C07315=1163.961,-99.989,-42.259,178.914,5.840,149.363
C07316=1163.967,-100.239,-42.250,178.911,5.839,149.364
C07317=1163.973,-100.489,-42.240,178.909,5.838,149.364
C07318=1163.977,-100.739,-42.231,178.907,5.838,149.365
C07319=1163.983,-100.989,-42.221,178.905,5.838,149.365
C07320=1163.988,-101.238,-42.212,178.903,5.838,149.366
C07321=1163.993,-101.488,-42.203,178.901,5.837,149.367
C07322=1163.999,-101.738,-42.193,178.899,5.837,149.367
C07323=1164.005,-102.010,-42.183,178.896,5.837,149.368
C07324=1164.011,-102.281,-42.173,178.894,5.836,149.368
C07325=1164.016,-102.553,-42.163,178.892,5.836,149.369
C07326=1164.022,-102.825,-42.153,178.890,5.836,149.370
C07327=1164.028,-103.075,-42.143,178.887,5.835,149.370
C07328=1164.033,-103.325,-42.134,178.885,5.835,149.371
C07329=1164.038,-103.574,-42.125,178.883,5.835,149.371
C07330=1164.044,-103.824,-42.115,178.881,5.834,149.372
C07331=1164.049,-104.074,-42.106,178.879,5.834,149.372
C07332=1164.054,-104.323,-42.097,178.877,5.834,149.373
C07333=1164.060,-104.574,-42.087,178.875,5.834,149.374
C07334=1164.065,-104.823,-42.078,178.873,5.833,149.374
C07335=1164.070,-105.073,-42.069,178.870,5.833,149.375
C07336=1164.076,-105.323,-42.059,178.868,5.833,149.375
C07337=1164.081,-105.573,-42.050,178.866,5.832,149.376
C07338=1164.086,-105.823,-42.041,178.864,5.833,149.376
C07339=1164.092,-106.073,-42.032,178.862,5.832,149.377
C07340=1164.097,-106.322,-42.022,178.860,5.832,149.377
C07341=1164.102,-106.572,-42.013,178.858,5.831,149.378
C07342=1164.107,-106.822,-42.004,178.856,5.831,149.379
C07343=1164.113,-107.072,-41.995,178.854,5.831,149.379
C07344=1164.118,-107.321,-41.985,178.851,5.830,149.380
C07345=1164.123,-107.571,-41.976,178.850,5.830,149.380
C07346=1164.128,-107.821,-41.968,178.847,5.830,149.381
C07347=1164.134,-108.071,-41.958,178.845,5.830,149.382
C07348=1164.140,-108.320,-41.950,178.843,5.829,149.382
C07349=1164.145,-108.570,-41.941,178.842,5.829,149.383
C07350=1164.150,-108.819,-41.931,178.839,5.829,149.383
C07351=1164.156,-109.069,-41.922,178.837,5.828,149.384
C07352=1164.161,-109.319,-41.913,178.835,5.828,149.384
C07353=1164.166,-109.569,-41.904,178.832,5.828,149.385
C07354=1164.171,-109.819,-41.895,178.831,5.828,149.385
C07355=1164.177,-110.069,-41.885,178.829,5.827,149.386
C07356=1164.182,-110.319,-41.876,178.827,5.827,149.387
C07357=1164.187,-110.568,-41.867,178.824,5.827,149.387
C07358=1164.192,-110.818,-41.858,178.823,5.827,149.388
C07359=1164.197,-111.068,-41.849,178.820,5.826,149.388
C07360=1164.204,-111.317,-41.840,178.819,5.826,149.389
C07361=1164.209,-111.567,-41.831,178.816,5.826,149.389
C07362=1164.214,-111.817,-41.822,178.814,5.825,149.390
C07363=1164.219,-112.067,-41.813,178.812,5.825,149.390
C07364=1164.225,-112.317,-41.804,178.810,5.824,149.391
C07365=1164.230,-112.567,-41.795,178.808,5.825,149.392
C07366=1164.236,-112.817,-41.786,178.806,5.824,149.392
C07367=1164.241,-113.067,-41.777,178.804,5.824,149.393
C07368=1164.246,-113.315,-41.768,178.802,5.823,149.393
C07369=1164.251,-113.565,-41.759,178.800,5.824,149.394
C07370=1164.257,-113.815,-41.750,178.798,5.823,149.394
C07371=1164.263,-114.065,-41.741,178.796,5.823,149.395
C07372=1164.268,-114.315,-41.732,178.793,5.823,149.396
C07373=1164.273,-114.565,-41.723,178.791,5.822,149.396
C07374=1164.278,-114.814,-41.714,178.789,5.822,149.396
C07375=1164.284,-115.064,-41.705,178.787,5.822,149.397
C07376=1164.289,-115.313,-41.696,178.785,5.822,149.398
C07377=1164.294,-115.563,-41.687,178.783,5.821,149.398
C07378=1164.299,-115.813,-41.679,178.781,5.821,149.399
C07379=1164.305,-116.063,-41.669,178.779,5.821,149.399
C07380=1164.310,-116.313,-41.660,178.777,5.821,149.400
C07381=1164.316,-116.562,-41.652,178.775,5.820,149.400
C07382=1164.322,-116.813,-41.643,178.773,5.820,149.401
C07383=1164.327,-117.063,-41.635,178.771,5.819,149.402
C07384=1164.332,-117.313,-41.626,178.769,5.820,149.402
C07385=1164.337,-117.562,-41.617,178.766,5.819,149.403
C07386=1164.342,-117.812,-41.608,178.765,5.819,149.403
C07387=1164.348,-118.061,-41.599,178.763,5.818,149.404
C07388=1164.353,-118.311,-41.590,178.761,5.818,149.404
C07389=1164.358,-118.561,-41.582,178.758,5.818,149.405
C07390=1164.364,-118.811,-41.573,178.757,5.818,149.405
C07391=1164.369,-119.061,-41.563,178.754,5.817,149.406
C07392=1164.375,-119.310,-41.555,178.752,5.818,149.407
C07393=1164.380,-119.560,-41.546,178.750,5.817,149.407
C07394=1164.386,-119.810,-41.537,178.748,5.816,149.408
C07395=1164.391,-120.060,-41.529,178.746,5.816,149.408
C07396=1164.396,-120.310,-41.520,178.744,5.816,149.409
C07397=1164.402,-120.559,-41.511,178.742,5.816,149.409
C07398=1164.407,-120.809,-41.502,178.740,5.815,149.410
C07399=1164.412,-121.059,-41.493,178.738,5.815,149.410
C07400=1164.417,-121.309,-41.485,178.736,5.815,149.411
C07401=1164.423,-121.558,-41.476,178.734,5.815,149.411
C07402=1164.429,-121.809,-41.468,178.732,5.814,149.412
C07403=1164.434,-122.058,-41.459,178.730,5.815,149.413
C07404=1164.439,-122.308,-41.450,178.728,5.814,149.413
C07405=1164.444,-122.558,-41.441,178.726,5.814,149.414
C07406=1164.450,-122.807,-41.433,178.724,5.813,149.414
C07407=1164.455,-123.058,-41.424,178.722,5.814,149.415
C07408=1164.461,-123.308,-41.416,178.720,5.813,149.415
C07409=1164.466,-123.557,-41.407,178.718,5.813,149.416
C07410=1164.471,-123.807,-41.398,178.716,5.812,149.416
C07411=1164.477,-124.056,-41.389,178.714,5.812,149.417
C07412=1164.482,-124.307,-41.381,178.711,5.812,149.418
C07413=1164.487,-124.556,-41.373,178.710,5.812,149.418
C07414=1164.492,-124.806,-41.364,178.708,5.811,149.418
C07415=1164.497,-125.055,-41.355,178.706,5.811,149.419
C07416=1164.503,-125.306,-41.347,178.703,5.811,149.420
C07417=1164.509,-125.555,-41.339,178.702,5.811,149.420
C07418=1164.514,-125.805,-41.330,178.700,5.810,149.421
C07419=1164.519,-126.055,-41.321,178.698,5.810,149.421
C07420=1164.525,-126.305,-41.313,178.695,5.810,149.422
C07421=1164.530,-126.554,-41.304,178.694,5.810,149.422
C07422=1164.535,-126.804,-41.295,178.692,5.809,149.423
C07423=1164.541,-127.055,-41.287,178.689,5.809,149.424
C07424=1164.547,-127.304,-41.278,178.687,5.809,149.424
C07425=1164.552,-127.554,-41.270,178.686,5.809,149.425
C07426=1164.557,-127.804,-41.262,178.683,5.808,149.425
C07427=1164.136,-127.815,-41.303,178.680,5.812,149.427
C07428=1164.130,-127.565,-41.311,178.682,5.812,149.426
C07429=1164.125,-127.315,-41.320,178.684,5.813,149.426
C07430=1164.119,-127.066,-41.329,178.686,5.812,149.425
C07431=1164.114,-126.815,-41.337,178.688,5.813,149.425
C07432=1164.109,-126.565,-41.346,178.690,5.813,149.424
C07433=1164.104,-126.316,-41.354,178.692,5.814,149.424
C07434=1164.098,-126.066,-41.362,178.694,5.813,149.423
C07435=1164.093,-125.816,-41.371,178.696,5.814,149.422
C07436=1164.088,-125.566,-41.380,178.698,5.814,149.422
C07437=1164.082,-125.317,-41.388,178.700,5.815,149.422
C07438=1164.077,-125.067,-41.396,178.702,5.815,149.421
C07439=1164.072,-124.817,-41.405,178.704,5.815,149.420
C07440=1164.066,-124.568,-41.414,178.706,5.815,149.420
C07441=1164.061,-124.318,-41.423,178.708,5.816,149.419
C07442=1164.055,-124.067,-41.431,178.710,5.816,149.419
C07443=1164.050,-123.818,-41.440,178.712,5.816,149.418
C07444=1164.044,-123.568,-41.448,178.714,5.816,149.418
C07445=1164.039,-123.319,-41.457,178.716,5.817,149.417
C07446=1164.034,-123.069,-41.466,178.718,5.817,149.417
C07447=1164.028,-122.818,-41.474,178.721,5.817,149.416
C07448=1164.023,-122.569,-41.483,178.722,5.817,149.415
C07449=1164.017,-122.319,-41.492,178.724,5.818,149.415
C07450=1164.012,-122.069,-41.501,178.726,5.817,149.414
C07451=1164.007,-121.819,-41.510,178.729,5.818,149.414
C07452=1164.001,-121.570,-41.517,178.730,5.818,149.413
C07453=1163.996,-121.320,-41.526,178.732,5.819,149.413
C07454=1163.991,-121.070,-41.535,178.734,5.818,149.412
C07455=1163.986,-120.820,-41.544,178.737,5.819,149.412
C07456=1163.980,-120.570,-41.553,178.738,5.819,149.411
C07457=1163.975,-120.321,-41.562,178.740,5.820,149.411
C07458=1163.969,-120.071,-41.570,178.743,5.820,149.410
C07459=1163.964,-119.821,-41.579,178.745,5.820,149.409
C07460=1163.959,-119.571,-41.587,178.746,5.820,149.409
C07461=1163.953,-119.322,-41.596,178.749,5.821,149.408
C07462=1163.948,-119.072,-41.605,178.751,5.821,149.408
C07463=1163.943,-118.822,-41.614,178.753,5.821,149.407
C07464=1163.938,-118.572,-41.623,178.754,5.821,149.407
C07465=1163.932,-118.322,-41.632,178.757,5.822,149.406
C07466=1163.927,-118.073,-41.641,178.759,5.822,149.406
C07467=1163.921,-117.823,-41.649,178.761,5.822,149.405
C07468=1163.916,-117.574,-41.658,178.762,5.822,149.405
C07469=1163.911,-117.323,-41.666,178.765,5.823,149.404
C07470=1163.906,-117.073,-41.675,178.767,5.824,149.403
C07471=1163.900,-116.823,-41.684,178.769,5.823,149.403
C07472=1163.894,-116.574,-41.693,178.772,5.824,149.402
C07473=1163.889,-116.324,-41.702,178.773,5.824,149.402
C07474=1163.884,-116.074,-41.711,178.775,5.825,149.401
C07475=1163.878,-115.824,-41.720,178.777,5.825,149.401
C07476=1163.873,-115.575,-41.729,178.780,5.825,149.400
C07477=1163.868,-115.325,-41.738,178.781,5.825,149.400
C07478=1163.862,-115.076,-41.746,178.783,5.826,149.399
C07479=1163.857,-114.826,-41.755,178.786,5.825,149.398
C07480=1163.851,-114.576,-41.764,178.788,5.826,149.398
C07481=1163.846,-114.326,-41.773,178.789,5.826,149.397
C07482=1163.841,-114.076,-41.782,178.792,5.826,149.397
C07483=1163.836,-113.826,-41.791,178.794,5.826,149.396
C07484=1163.831,-113.576,-41.800,178.796,5.827,149.396
C07485=1163.825,-113.327,-41.809,178.797,5.827,149.395
C07486=1163.820,-113.077,-41.817,178.800,5.827,149.394
C07487=1163.814,-112.827,-41.827,178.802,5.828,149.394
C07488=1163.809,-112.577,-41.836,178.804,5.828,149.393
C07489=1163.803,-112.327,-41.845,178.807,5.829,149.393
C07490=1163.799,-112.078,-41.854,178.808,5.828,149.392
C07491=1163.793,-111.828,-41.863,178.810,5.829,149.392
C07492=1163.788,-111.578,-41.872,178.812,5.829,149.391
C07493=1163.782,-111.329,-41.881,178.815,5.830,149.391
C07494=1163.777,-111.079,-41.890,178.816,5.830,149.390
C07495=1163.771,-110.829,-41.899,178.819,5.830,149.389
C07496=1163.766,-110.579,-41.908,178.821,5.830,149.389
C07497=1163.761,-110.329,-41.917,178.823,5.831,149.388
C07498=1163.755,-110.079,-41.926,178.825,5.831,149.388
C07499=1163.750,-109.829,-41.935,178.827,5.831,149.387
C07500=1163.745,-109.580,-41.945,178.829,5.832,149.387
C07501=1163.740,-109.330,-41.954,178.831,5.832,149.386
C07502=1163.734,-109.080,-41.963,178.833,5.832,149.386
C07503=1163.729,-108.830,-41.972,178.835,5.832,149.385
C07504=1163.723,-108.581,-41.981,178.837,5.833,149.385
C07505=1163.718,-108.331,-41.990,178.839,5.832,149.384
C07506=1163.712,-108.082,-42.000,178.842,5.833,149.383
C07507=1163.707,-107.832,-42.009,178.844,5.834,149.383
C07508=1163.702,-107.582,-42.018,178.846,5.834,149.382
C07509=1163.697,-107.332,-42.027,178.848,5.834,149.382
C07510=1163.691,-107.082,-42.036,178.850,5.834,149.381
C07511=1163.686,-106.833,-42.046,178.852,5.835,149.380
C07512=1163.681,-106.583,-42.055,178.854,5.835,149.380
C07513=1163.676,-106.333,-42.063,178.856,5.835,149.380
C07514=1163.670,-106.083,-42.073,178.859,5.836,149.379
C07515=1163.665,-105.833,-42.082,178.860,5.836,149.378
C07516=1163.660,-105.584,-42.091,178.863,5.837,149.378
C07517=1163.654,-105.334,-42.101,178.865,5.836,149.377
C07518=1163.649,-105.084,-42.110,178.867,5.837,149.377
C07519=1163.644,-104.834,-42.119,178.868,5.837,149.376
C07520=1163.639,-104.585,-42.128,178.871,5.837,149.375
C07521=1163.633,-104.335,-42.138,178.873,5.838,149.375
C07522=1163.628,-104.085,-42.147,178.875,5.838,149.374
C07523=1163.623,-103.836,-42.156,178.878,5.838,149.374
C07524=1163.617,-103.585,-42.166,178.879,5.838,149.373
C07525=1163.612,-103.336,-42.175,178.882,5.839,149.373
C07526=1163.607,-103.086,-42.184,178.883,5.839,149.372
C07527=1163.601,-102.836,-42.194,178.886,5.839,149.372
C07528=1163.596,-102.564,-42.204,178.888,5.840,149.371
C07529=1163.589,-102.292,-42.213,178.890,5.840,149.370
C07530=1163.584,-102.020,-42.223,178.893,5.840,149.370
C07531=1163.577,-101.748,-42.234,178.895,5.841,149.369
C07532=1163.573,-101.499,-42.244,178.897,5.840,149.368
C07533=1163.567,-101.249,-42.253,178.899,5.841,149.368
C07534=1163.561,-100.999,-42.262,178.902,5.842,149.367
C07535=1163.557,-100.750,-42.272,178.903,5.842,149.367
C07536=1163.551,-100.500,-42.281,178.905,5.842,149.366
C07537=1163.546,-100.250,-42.290,178.908,5.842,149.366
C07538=1163.541,-100.001,-42.300,178.910,5.843,149.365
C07539=1163.535,-99.750,-42.309,178.912,5.844,149.365
C07540=1163.530,-99.501,-42.319,178.914,5.843,149.364
C07541=1163.525,-99.251,-42.328,178.916,5.844,149.363
C07542=1163.519,-99.001,-42.337,178.918,5.843,149.363
C07543=1163.514,-98.752,-42.347,178.920,5.844,149.362
C07544=1163.508,-98.502,-42.356,178.923,5.845,149.362
C07545=1163.504,-98.252,-42.366,178.925,5.845,149.361
C07546=1163.498,-98.002,-42.376,178.927,5.845,149.361
C07547=1163.493,-97.752,-42.386,178.929,5.845,149.360
C07548=1163.487,-97.502,-42.395,178.931,5.846,149.359
C07549=1163.482,-97.253,-42.405,178.933,5.846,149.359
C07550=1163.476,-97.003,-42.414,178.935,5.846,149.358
C07551=1163.471,-96.753,-42.423,178.938,5.847,149.358
C07552=1163.466,-96.504,-42.433,178.939,5.847,149.357
C07553=1163.460,-96.254,-42.442,178.942,5.847,149.356
C07554=1163.456,-96.004,-42.452,178.944,5.848,149.356
C07555=1163.450,-95.754,-42.461,178.946,5.848,149.356
C07556=1163.445,-95.505,-42.471,178.948,5.848,149.355
C07557=1163.439,-95.255,-42.480,178.950,5.848,149.354
C07558=1163.435,-95.005,-42.490,178.953,5.849,149.354
C07559=1163.429,-94.755,-42.500,178.955,5.849,149.353
C07560=1163.424,-94.505,-42.509,178.956,5.849,149.353
C07561=1163.418,-94.256,-42.520,178.959,5.850,149.352
C07562=1163.413,-94.006,-42.529,178.961,5.850,149.351
C07563=1163.408,-93.757,-42.539,178.963,5.850,149.351
C07564=1163.402,-93.506,-42.548,178.966,5.851,149.350
C07565=1163.397,-93.257,-42.558,178.967,5.851,149.350
C07566=1163.391,-93.007,-42.567,178.970,5.851,149.349
C07567=1163.387,-92.757,-42.577,178.972,5.852,149.349
C07568=1163.381,-92.507,-42.587,178.974,5.852,149.348
C07569=1163.376,-92.258,-42.596,178.976,5.852,149.347
C07570=1163.370,-92.008,-42.607,178.978,5.852,149.347
C07571=1163.365,-91.758,-42.616,178.981,5.853,149.346
C07572=1163.359,-91.509,-42.626,178.983,5.854,149.346
C07573=1163.354,-91.258,-42.636,178.985,5.853,149.345
C07574=1163.349,-91.009,-42.645,178.987,5.854,149.344
C07575=1163.344,-90.759,-42.655,178.989,5.855,149.344
C07576=1163.339,-90.509,-42.664,178.991,5.854,149.343
C07577=1163.333,-90.260,-42.675,178.994,5.855,149.343
C07578=1163.328,-90.010,-42.684,178.996,5.855,149.342
C07579=1163.323,-89.760,-42.694,178.998,5.855,149.342
C07580=1163.317,-89.510,-42.704,179.000,5.856,149.341
C07581=1163.312,-89.261,-42.714,179.002,5.856,149.340
C07582=1163.306,-89.011,-42.723,179.004,5.857,149.340
C07583=1163.301,-88.761,-42.734,179.007,5.857,149.339
C07584=1163.296,-88.512,-42.743,179.009,5.857,149.339
C07585=1163.291,-88.262,-42.754,179.011,5.858,149.338
C07586=1163.286,-88.012,-42.763,179.013,5.857,149.338
C07587=1163.280,-87.762,-42.773,179.015,5.858,149.337
C07588=1163.275,-87.513,-42.783,179.018,5.858,149.336
C07589=1163.269,-87.263,-42.792,179.019,5.858,149.336
C07590=1163.264,-87.013,-42.803,179.022,5.859,149.335
C07591=1163.259,-86.763,-42.813,179.024,5.860,149.335
C07592=1163.254,-86.514,-42.822,179.026,5.860,149.334
C07593=1163.248,-86.264,-42.832,179.028,5.860,149.333
C07594=1163.243,-86.013,-42.842,179.031,5.861,149.333
C07595=1163.238,-85.764,-42.852,179.033,5.860,149.332
C07596=1163.233,-85.515,-42.862,179.035,5.861,149.332
C07597=1163.227,-85.264,-42.872,179.037,5.862,149.331
C07598=1163.222,-85.015,-42.882,179.039,5.861,149.331
C07599=1163.217,-84.765,-42.892,179.041,5.862,149.330
C07600=1163.211,-84.515,-42.902,179.044,5.863,149.329
C07601=1163.206,-84.266,-42.912,179.046,5.863,149.329
C07602=1163.201,-84.016,-42.922,179.048,5.863,149.328
C07603=1163.195,-83.766,-42.932,179.050,5.864,149.328
C07604=1163.190,-83.516,-42.942,179.052,5.864,149.327
C07605=1163.185,-83.267,-42.952,179.055,5.864,149.327
C07606=1163.180,-83.017,-42.962,179.057,5.865,149.326
C07607=1163.174,-82.767,-42.972,179.059,5.865,149.325
C07608=1163.169,-82.518,-42.983,179.061,5.865,149.325
C07609=1163.164,-82.268,-42.992,179.064,5.866,149.324
C07610=1163.159,-82.018,-43.002,179.065,5.866,149.324
C07611=1163.153,-81.768,-43.012,179.068,5.866,149.323
C07612=1163.147,-81.519,-43.023,179.070,5.867,149.323
C07613=1163.143,-81.269,-43.033,179.072,5.867,149.322
C07614=1163.138,-81.019,-43.043,179.075,5.867,149.321
C07615=1163.132,-80.769,-43.053,179.077,5.868,149.321
C07616=1163.126,-80.520,-43.063,179.079,5.868,149.320
C07617=1163.122,-80.270,-43.073,179.081,5.868,149.320
C07618=1163.117,-80.020,-43.083,179.084,5.869,149.319
C07619=1163.111,-79.771,-43.094,179.085,5.869,149.318
C07620=1163.106,-79.520,-43.103,179.088,5.870,149.318
C07621=1163.100,-79.271,-43.114,179.090,5.870,149.317
C07622=1163.094,-79.021,-43.124,179.092,5.870,149.317
C07623=1163.090,-78.771,-43.134,179.094,5.870,149.316
C07624=1163.085,-78.522,-43.144,179.097,5.871,149.316
C07625=1163.079,-78.272,-43.154,179.099,5.871,149.315
C07626=1163.074,-78.022,-43.165,179.101,5.871,149.314
C07627=1163.068,-77.772,-43.175,179.104,5.872,149.314
C07628=1163.063,-77.523,-43.185,179.105,5.872,149.313
C07629=1163.059,-77.273,-43.195,179.107,5.873,149.313
C07630=1163.053,-77.023,-43.205,179.110,5.873,149.312
C07631=1163.047,-76.774,-43.216,179.112,5.873,149.312
C07632=1163.041,-76.502,-43.227,179.114,5.873,149.311
C07633=1163.036,-76.231,-43.238,179.117,5.874,149.310
C07634=1163.030,-75.960,-43.249,179.119,5.875,149.310
C07635=1163.025,-75.689,-43.261,179.122,5.875,149.309
C07636=1163.019,-75.440,-43.271,179.124,5.875,149.308
C07637=1163.014,-75.189,-43.282,179.126,5.875,149.308
C07638=1163.009,-74.940,-43.292,179.128,5.876,149.307
C07639=1163.003,-74.690,-43.302,179.131,5.877,149.307
C07640=1162.998,-74.440,-43.313,179.133,5.877,149.306
C07641=1162.992,-74.190,-43.323,179.135,5.877,149.305
C07642=1162.987,-73.940,-43.333,179.137,5.878,149.305
C07643=1162.982,-73.691,-43.344,179.139,5.877,149.304
C07644=1162.976,-73.441,-43.354,179.142,5.878,149.304
C07645=1162.971,-73.191,-43.364,179.144,5.878,149.303
C07646=1162.967,-72.942,-43.375,179.146,5.878,149.303
C07647=1162.961,-72.693,-43.385,179.149,5.879,149.302
C07648=1162.956,-72.442,-43.396,179.151,5.880,149.301
C07649=1162.951,-72.193,-43.406,179.153,5.880,149.301
C07650=1162.946,-71.943,-43.416,179.155,5.880,149.300
C07651=1162.940,-71.693,-43.427,179.157,5.881,149.300
C07652=1162.935,-71.443,-43.437,179.160,5.881,149.299
C07653=1162.930,-71.194,-43.448,179.162,5.881,149.298
C07654=1162.924,-70.944,-43.458,179.164,5.882,149.298
C07655=1162.919,-70.694,-43.469,179.166,5.882,149.297
C07656=1162.913,-70.445,-43.479,179.169,5.883,149.297
C07657=1162.908,-70.194,-43.490,179.171,5.883,149.296
C07658=1162.903,-69.945,-43.501,179.173,5.883,149.295
C07659=1162.898,-69.695,-43.511,179.176,5.884,149.295
C07660=1162.893,-69.446,-43.521,179.178,5.884,149.294
C07661=1162.887,-69.196,-43.532,179.180,5.884,149.294
C07662=1162.882,-68.947,-43.543,179.182,5.885,149.293
C07663=1162.877,-68.697,-43.553,179.185,5.885,149.293
C07664=1162.872,-68.447,-43.564,179.187,5.885,149.292
C07665=1162.866,-68.197,-43.574,179.189,5.886,149.291
C07666=1162.861,-67.948,-43.585,179.192,5.886,149.291
C07667=1162.855,-67.698,-43.596,179.194,5.887,149.290
C07668=1162.850,-67.447,-43.606,179.195,5.887,149.290
C07669=1162.844,-67.198,-43.617,179.198,5.887,149.289
C07670=1162.840,-66.948,-43.628,179.200,5.888,149.288
C07671=1162.834,-66.699,-43.638,179.202,5.888,149.288
C07672=1162.829,-66.449,-43.649,179.204,5.889,149.287
C07673=1162.824,-66.200,-43.660,179.207,5.889,149.287
C07674=1162.819,-65.949,-43.670,179.209,5.890,149.286
C07675=1162.813,-65.700,-43.680,179.211,5.889,149.285
C07676=1162.809,-65.450,-43.692,179.214,5.890,149.285
C07677=1162.803,-65.201,-43.702,179.216,5.891,149.284
C07678=1162.798,-64.950,-43.713,179.218,5.891,149.284
C07679=1162.793,-64.701,-43.723,179.221,5.891,149.283
C07680=1162.787,-64.451,-43.735,179.223,5.892,149.283
C07681=1162.782,-64.202,-43.746,179.225,5.892,149.282
C07682=1162.777,-63.952,-43.756,179.228,5.893,149.281
C07683=1162.771,-63.702,-43.766,179.230,5.893,149.281
C07684=1162.766,-63.453,-43.778,179.232,5.893,149.280
C07685=1162.761,-63.203,-43.788,179.235,5.894,149.279
C07686=1162.756,-62.953,-43.799,179.237,5.895,149.279
C07687=1162.750,-62.704,-43.810,179.239,5.894,149.278
C07688=1162.745,-62.453,-43.821,179.241,5.895,149.278
C07689=1162.740,-62.204,-43.832,179.244,5.895,149.277
C07690=1162.734,-61.954,-43.842,179.246,5.896,149.277
C07691=1162.730,-61.705,-43.853,179.248,5.896,149.276
C07692=1162.724,-61.455,-43.864,179.250,5.897,149.275
C07693=1162.719,-61.205,-43.875,179.253,5.897,149.275
C07694=1162.713,-60.955,-43.886,179.255,5.898,149.274
C07695=1162.708,-60.706,-43.897,179.257,5.897,149.274
C07696=1162.703,-60.456,-43.907,179.259,5.898,149.273
C07697=1162.698,-60.207,-43.918,179.262,5.899,149.272
C07698=1162.693,-59.956,-43.929,179.264,5.899,149.272
C07699=1162.687,-59.707,-43.940,179.267,5.900,149.271
C07700=1162.682,-59.457,-43.951,179.268,5.900,149.271
C07701=1162.677,-59.207,-43.962,179.271,5.900,149.270
C07702=1162.672,-58.958,-43.973,179.273,5.901,149.270
C07703=1162.666,-58.708,-43.984,179.276,5.901,149.269
C07704=1162.661,-58.458,-43.995,179.277,5.901,149.268
C07705=1162.656,-58.209,-44.006,179.280,5.902,149.268
C07706=1162.651,-57.958,-44.017,179.282,5.903,149.267
C07707=1162.645,-57.709,-44.028,179.285,5.903,149.266
C07708=1162.640,-57.460,-44.039,179.287,5.903,149.266
C07709=1162.635,-57.210,-44.050,179.289,5.903,149.265
C07710=1162.630,-56.960,-44.061,179.291,5.904,149.265
C07711=1162.624,-56.710,-44.072,179.294,5.905,149.264
C07712=1162.619,-56.461,-44.083,179.296,5.905,149.264
C07713=1162.614,-56.211,-44.094,179.298,5.905,149.263
C07714=1162.609,-55.961,-44.105,179.300,5.906,149.262
C07715=1162.603,-55.712,-44.116,179.303,5.906,149.262
C07716=1162.598,-55.462,-44.127,179.305,5.907,149.261
C07717=1162.594,-55.212,-44.138,179.308,5.907,149.261
C07718=1162.588,-54.963,-44.150,179.310,5.907,149.260
C07719=1162.583,-54.712,-44.160,179.312,5.908,149.259
C07720=1162.578,-54.463,-44.172,179.314,5.909,149.259
C07721=1162.572,-54.214,-44.183,179.317,5.909,149.258
C07722=1162.567,-53.963,-44.194,179.319,5.910,149.258
C07723=1162.562,-53.714,-44.205,179.321,5.909,149.257
C07724=1162.556,-53.465,-44.216,179.324,5.910,149.257
C07725=1162.551,-53.215,-44.228,179.326,5.911,149.256
C07726=1162.546,-52.965,-44.238,179.328,5.911,149.255
C07727=1162.540,-52.715,-44.250,179.331,5.912,149.255
C07728=1162.536,-52.466,-44.261,179.333,5.912,149.254
C07729=1162.531,-52.216,-44.272,179.335,5.912,149.253
C07730=1162.525,-51.966,-44.284,179.338,5.913,149.253
C07731=1162.520,-51.717,-44.295,179.340,5.913,149.252
C07732=1162.515,-51.467,-44.306,179.342,5.914,149.252
C07733=1162.510,-51.216,-44.317,179.344,5.914,149.251
C07734=1162.504,-50.968,-44.328,179.347,5.914,149.250
C07735=1162.499,-50.718,-44.340,179.349,5.915,149.250
C07736=1162.493,-50.447,-44.352,179.352,5.915,149.249
C07737=1162.488,-50.177,-44.363,179.354,5.916,149.249
C07738=1162.483,-49.906,-44.376,179.357,5.917,149.248
C07739=1162.477,-49.635,-44.389,179.360,5.917,149.247
C07740=1162.471,-49.386,-44.400,179.362,5.918,149.247
C07741=1162.466,-49.137,-44.411,179.364,5.917,149.246
C07742=1162.461,-48.887,-44.423,179.366,5.918,149.245
C07743=1162.456,-48.636,-44.434,179.369,5.919,149.245
C07744=1162.450,-48.387,-44.445,179.371,5.919,149.244
C07745=1162.445,-48.137,-44.457,179.373,5.920,149.244
C07746=1162.440,-47.888,-44.468,179.376,5.920,149.243
C07747=1162.435,-47.638,-44.480,179.378,5.920,149.243
C07748=1162.430,-47.389,-44.491,179.380,5.921,149.242
C07749=1162.424,-47.139,-44.503,179.383,5.921,149.241
C07750=1162.419,-46.889,-44.513,179.385,5.922,149.241
C07751=1162.414,-46.639,-44.525,179.387,5.923,149.240
C07752=1162.408,-46.390,-44.536,179.390,5.923,149.240
C07753=1162.403,-46.140,-44.548,179.392,5.923,149.239
C07754=1162.398,-45.890,-44.559,179.394,5.923,149.238
C07755=1162.393,-45.640,-44.571,179.397,5.924,149.238
C07756=1162.388,-45.391,-44.582,179.399,5.925,149.237
C07757=1162.382,-45.142,-44.594,179.401,5.925,149.237
C07758=1162.377,-44.892,-44.605,179.404,5.926,149.236
C07759=1162.372,-44.642,-44.617,179.406,5.926,149.236
C07760=1162.367,-44.392,-44.628,179.408,5.926,149.235
C07761=1162.362,-44.142,-44.640,179.410,5.927,149.234
C07762=1162.356,-43.893,-44.652,179.413,5.928,149.234
C07763=1162.351,-43.644,-44.663,179.416,5.928,149.233
C07764=1162.346,-43.394,-44.675,179.418,5.929,149.232
C07765=1162.341,-43.144,-44.686,179.421,5.929,149.232
C07766=1162.336,-42.894,-44.698,179.422,5.929,149.231
C07767=1162.331,-42.644,-44.709,179.425,5.930,149.231
C07768=1162.325,-42.395,-44.721,179.427,5.930,149.230
C07769=1162.320,-42.145,-44.733,179.430,5.931,149.229
C07770=1162.315,-41.896,-44.744,179.432,5.932,149.229
C07771=1162.309,-41.646,-44.756,179.435,5.932,149.228
C07772=1162.305,-41.396,-44.767,179.437,5.933,149.228
C07773=1162.299,-41.146,-44.779,179.439,5.932,149.227
C07774=1162.293,-40.897,-44.791,179.441,5.933,149.227
C07775=1162.289,-40.647,-44.802,179.444,5.934,149.226
C07776=1162.283,-40.397,-44.814,179.446,5.934,149.225
C07777=1162.278,-40.147,-44.826,179.449,5.935,149.225
C07778=1162.273,-39.898,-44.837,179.451,5.935,149.224
C07779=1162.268,-39.648,-44.850,179.453,5.936,149.224
C07780=1162.263,-39.399,-44.861,179.455,5.936,149.223
C07781=1162.258,-39.149,-44.873,179.458,5.937,149.222
C07782=1162.252,-38.900,-44.884,179.460,5.937,149.222
C07783=1162.247,-38.650,-44.896,179.463,5.938,149.221
C07784=1162.242,-38.400,-44.907,179.465,5.938,149.220
C07785=1162.236,-38.150,-44.919,179.467,5.939,149.220
C07786=1162.231,-37.901,-44.932,179.470,5.939,149.219
C07787=1162.226,-37.651,-44.943,179.472,5.940,149.219
C07788=1162.221,-37.401,-44.955,179.474,5.940,149.218
C07789=1162.215,-37.151,-44.967,179.476,5.941,149.218
C07790=1162.211,-36.902,-44.978,179.479,5.941,149.217
C07791=1162.206,-36.652,-44.991,179.482,5.941,149.216
C07792=1162.200,-36.403,-45.002,179.484,5.942,149.216
C07793=1162.194,-36.153,-45.014,179.487,5.943,149.215
C07794=1162.190,-35.904,-45.026,179.489,5.943,149.215
C07795=1162.184,-35.654,-45.037,179.492,5.944,149.214
C07796=1162.179,-35.404,-45.050,179.494,5.945,149.213
C07797=1162.174,-35.155,-45.061,179.496,5.944,149.213
C07798=1162.169,-34.905,-45.073,179.498,5.945,149.212
C07799=1162.163,-34.655,-45.085,179.501,5.946,149.212
C07800=1162.158,-34.406,-45.098,179.503,5.946,149.211
C07801=1162.153,-34.156,-45.110,179.505,5.947,149.210
C07802=1162.148,-33.906,-45.121,179.508,5.947,149.210
C07803=1162.143,-33.657,-45.134,179.510,5.948,149.209
C07804=1162.138,-33.407,-45.145,179.513,5.948,149.209
C07805=1162.132,-33.157,-45.157,179.515,5.949,149.208
C07806=1162.128,-32.908,-45.169,179.517,5.949,149.207
C07807=1162.122,-32.658,-45.181,179.519,5.950,149.207
C07808=1162.117,-32.408,-45.193,179.522,5.950,149.206
C07809=1162.112,-32.159,-45.206,179.524,5.951,149.206
C07810=1162.106,-31.909,-45.218,179.527,5.951,149.205
C07811=1162.101,-31.659,-45.229,179.529,5.952,149.205
C07812=1162.097,-31.410,-45.241,179.532,5.953,149.204
C07813=1162.091,-31.160,-45.253,179.534,5.953,149.203
C07814=1162.086,-30.910,-45.265,179.537,5.954,149.203
C07815=1162.081,-30.661,-45.278,179.539,5.954,149.202
C07816=1162.075,-30.411,-45.290,179.541,5.955,149.202
C07817=1162.070,-30.161,-45.302,179.544,5.955,149.201
C07818=1162.065,-29.912,-45.314,179.546,5.955,149.200
C07819=1162.060,-29.662,-45.325,179.548,5.956,149.200
C07820=1162.055,-29.412,-45.338,179.551,5.957,149.199
C07821=1162.049,-29.162,-45.350,179.553,5.957,149.198
C07822=1162.044,-28.913,-45.363,179.555,5.958,149.198
C07823=1162.039,-28.663,-45.374,179.558,5.958,149.197
C07824=1162.034,-28.414,-45.387,179.561,5.959,149.197
C07825=1162.028,-28.164,-45.399,179.563,5.960,149.196
C07826=1162.024,-27.915,-45.411,179.566,5.960,149.195
C07827=1162.018,-27.665,-45.423,179.568,5.961,149.195
C07828=1162.013,-27.416,-45.435,179.570,5.961,149.194
C07829=1162.008,-27.166,-45.447,179.573,5.962,149.194
C07830=1162.003,-26.916,-45.460,179.575,5.962,149.193
C07831=1161.998,-26.666,-45.472,179.577,5.962,149.193
C07832=1161.993,-26.416,-45.485,179.579,5.963,149.192
C07833=1161.987,-26.167,-45.497,179.582,5.964,149.191
C07834=1161.982,-25.917,-45.509,179.584,5.964,149.191
C07835=1161.977,-25.667,-45.521,179.587,5.965,149.190
C07836=1161.972,-25.418,-45.534,179.589,5.965,149.190
C07837=1161.966,-25.168,-45.546,179.592,5.966,149.189
C07838=1161.961,-24.919,-45.558,179.594,5.967,149.188
C07839=1161.956,-24.669,-45.571,179.597,5.967,149.188
C07840=1161.951,-24.399,-45.584,179.599,5.967,149.187
C07841=1161.946,-24.129,-45.597,179.601,5.968,149.187
C07842=1161.939,-23.859,-45.611,179.604,5.969,149.186
C07843=1161.934,-23.589,-45.624,179.607,5.969,149.185
C07844=1161.929,-23.340,-45.636,179.609,5.970,149.185
C07845=1161.924,-23.090,-45.649,179.612,5.970,149.184
C07846=1161.918,-22.840,-45.661,179.614,5.971,149.184
C07847=1161.913,-22.591,-45.673,179.616,5.972,149.183
C07848=1161.908,-22.342,-45.686,179.619,5.972,149.182
C07849=1161.903,-22.091,-45.698,179.621,5.973,149.182
C07850=1161.898,-21.842,-45.711,179.624,5.973,149.181
C07851=1161.893,-21.593,-45.723,179.626,5.974,149.181
C07852=1161.887,-21.343,-45.735,179.629,5.975,149.180
C07853=1161.882,-21.093,-45.748,179.631,5.975,149.179
C07854=1161.877,-20.844,-45.760,179.634,5.976,149.179
C07855=1161.872,-20.594,-45.772,179.636,5.977,149.178
C07856=1161.866,-20.344,-45.786,179.639,5.977,149.177
C07857=1161.861,-20.094,-45.798,179.641,5.977,149.177
C07858=1161.856,-19.845,-45.811,179.643,5.978,149.176
C07859=1161.851,-19.595,-45.823,179.646,5.979,149.176
C07860=1161.846,-19.346,-45.836,179.648,5.980,149.175
C07861=1161.841,-19.096,-45.849,179.651,5.980,149.174
C07862=1161.836,-18.846,-45.861,179.653,5.981,149.174
C07863=1161.831,-18.597,-45.873,179.656,5.981,149.173
C07864=1161.825,-18.347,-45.886,179.658,5.982,149.173
C07865=1161.820,-18.098,-45.898,179.661,5.982,149.172
C07866=1161.815,-17.848,-45.912,179.663,5.983,149.171
C07867=1161.810,-17.598,-45.924,179.665,5.984,149.171
C07868=1161.804,-17.348,-45.936,179.668,5.984,149.170
C07869=1161.799,-17.099,-45.949,179.670,5.985,149.170
C07870=1161.794,-16.850,-45.961,179.673,5.985,149.169
C07871=1161.790,-16.600,-45.974,179.675,5.986,149.169
C07872=1161.784,-16.350,-45.988,179.678,5.987,149.168
C07873=1161.779,-16.101,-46.000,179.680,5.987,149.167
C07874=1161.774,-15.851,-46.013,179.683,5.988,149.167
C07875=1161.769,-15.601,-46.025,179.685,5.988,149.166
C07876=1161.764,-15.351,-46.038,179.687,5.989,149.166
C07877=1161.758,-15.102,-46.051,179.690,5.990,149.165
C07878=1161.753,-14.853,-46.063,179.692,5.990,149.164
C07879=1161.748,-14.602,-46.076,179.695,5.991,149.164
C07880=1161.743,-14.353,-46.089,179.697,5.992,149.163
C07881=1161.738,-14.104,-46.102,179.700,5.992,149.163
C07882=1161.732,-13.854,-46.115,179.702,5.993,149.162
C07883=1161.727,-13.604,-46.128,179.705,5.993,149.161
C07884=1161.722,-13.355,-46.140,179.707,5.994,149.161
C07885=1161.717,-13.106,-46.153,179.709,5.995,149.160
C07886=1161.711,-12.856,-46.166,179.712,5.995,149.160
C07887=1161.707,-12.606,-46.179,179.714,5.996,149.159
C07888=1161.701,-12.356,-46.191,179.717,5.996,149.158
C07889=1161.696,-12.107,-46.204,179.719,5.997,149.158
C07890=1161.691,-11.856,-46.217,179.722,5.998,149.157
C07891=1161.686,-11.607,-46.230,179.724,5.998,149.157
C07892=1161.681,-11.358,-46.242,179.727,5.999,149.156
C07893=1161.677,-11.108,-46.256,179.729,5.999,149.155
C07894=1161.671,-10.859,-46.269,179.731,6.000,149.155
C07895=1161.666,-10.609,-46.282,179.734,6.001,149.154
C07896=1161.661,-10.359,-46.295,179.736,6.001,149.154
C07897=1161.655,-10.110,-46.308,179.739,6.002,149.153
C07898=1161.650,-9.860,-46.321,179.741,6.003,149.153
C07899=1161.646,-9.610,-46.334,179.744,6.003,149.152
C07900=1161.640,-9.361,-46.347,179.746,6.004,149.151
C07901=1161.635,-9.111,-46.359,179.749,6.004,149.151
C07902=1161.630,-8.861,-46.372,179.751,6.005,149.150
C07903=1161.624,-8.612,-46.386,179.753,6.006,149.150
C07904=1161.619,-8.362,-46.398,179.756,6.006,149.149
C07905=1161.615,-8.112,-46.411,179.758,6.007,149.148
C07906=1161.609,-7.863,-46.425,179.761,6.007,149.148
C07907=1161.604,-7.614,-46.438,179.763,6.008,149.147
C07908=1161.599,-7.364,-46.451,179.766,6.009,149.147
C07909=1161.593,-7.114,-46.464,179.768,6.009,149.146
C07910=1161.589,-6.864,-46.477,179.771,6.010,149.145
C07911=1161.583,-6.615,-46.490,179.773,6.010,149.145
C07912=1161.578,-6.366,-46.503,179.776,6.012,149.144
C07913=1161.574,-6.116,-46.516,179.779,6.012,149.144
C07914=1161.568,-5.866,-46.529,179.781,6.013,149.143
C07915=1161.563,-5.617,-46.542,179.783,6.014,149.142
C07916=1161.558,-5.367,-46.556,179.786,6.014,149.142
C07917=1161.552,-5.118,-46.568,179.788,6.015,149.141
C07918=1161.548,-4.868,-46.582,179.790,6.016,149.141
C07919=1161.542,-4.618,-46.595,179.793,6.016,149.140
C07920=1161.538,-4.368,-46.608,179.796,6.017,149.139
C07921=1161.532,-4.119,-46.621,179.798,6.017,149.139
C07922=1161.527,-3.870,-46.635,179.801,6.018,149.138
C07923=1161.522,-3.620,-46.648,179.803,6.019,149.138
C07924=1161.517,-3.370,-46.661,179.805,6.019,149.137
C07925=1161.512,-3.121,-46.675,179.808,6.020,149.137
C07926=1161.507,-2.871,-46.688,179.810,6.020,149.136
C07927=1161.501,-2.621,-46.701,179.812,6.021,149.136
C07928=1161.496,-2.372,-46.714,179.816,6.022,149.135
C07929=1161.491,-2.123,-46.728,179.818,6.023,149.134
C07930=1161.486,-1.873,-46.741,179.820,6.024,149.134
C07931=1161.480,-1.623,-46.754,179.823,6.024,149.133
C07932=1161.476,-1.374,-46.768,179.825,6.025,149.133
C07933=1161.470,-1.124,-46.781,179.828,6.025,149.132
C07934=1161.466,-0.874,-46.794,179.830,6.026,149.131
C07935=1161.460,-0.625,-46.808,179.833,6.027,149.131
C07936=1161.456,-0.375,-46.821,179.835,6.028,149.130
C07937=1161.450,-0.126,-46.835,179.838,6.028,149.130
C07938=1161.446,0.124,-46.847,179.840,6.029,149.129
C07939=1161.440,0.374,-46.861,179.842,6.029,149.128
C07940=1161.435,0.623,-46.875,179.845,6.030,149.128
C07941=1161.430,0.873,-46.888,179.848,6.031,149.127
C07942=1161.425,1.122,-46.902,179.851,6.032,149.127
C07943=1161.420,1.372,-46.914,179.853,6.033,149.126
C07944=1161.414,1.641,-46.929,179.855,6.033,149.125
C07945=1161.408,1.911,-46.944,179.858,6.034,149.125
C07946=1161.402,2.180,-46.958,179.861,6.035,149.124
C07947=1161.398,2.449,-46.973,179.863,6.036,149.124
C07948=1161.392,2.699,-46.986,179.866,6.036,149.123
C07949=1161.387,2.948,-47.000,179.868,6.037,149.122
C07950=1161.382,3.198,-47.013,179.871,6.037,149.122
C07951=1161.377,3.447,-47.027,179.873,6.038,149.121
C07952=1161.371,3.698,-47.041,179.876,6.039,149.121
C07953=1161.367,3.946,-47.054,179.878,6.039,149.120
C07954=1161.361,4.197,-47.068,179.881,6.041,149.119
C07955=1161.356,4.446,-47.081,179.884,6.041,149.119
C07956=1161.351,4.696,-47.094,179.886,6.042,149.118
C07957=1161.346,4.945,-47.109,179.889,6.042,149.118
C07958=1161.341,5.194,-47.123,179.891,6.043,149.117
C07959=1161.336,5.444,-47.136,179.893,6.044,149.116
C07960=1161.331,5.693,-47.149,179.896,6.045,149.116
C07961=1161.325,5.944,-47.163,179.898,6.045,149.115
C07962=1161.321,6.192,-47.176,179.901,6.047,149.115
C07963=1161.316,6.442,-47.191,179.904,6.047,149.114
C07964=1161.310,6.692,-47.204,179.906,6.048,149.113
C07965=1161.306,6.941,-47.217,179.909,6.048,149.113
C07966=1161.300,7.191,-47.231,179.911,6.049,149.112
C07967=1161.295,7.440,-47.245,179.913,6.050,149.112
C07968=1161.290,7.690,-47.259,179.916,6.050,149.111
C07969=1161.285,7.940,-47.272,179.918,6.051,149.111
C07970=1161.280,8.189,-47.286,179.921,6.052,149.110
C07971=1161.275,8.439,-47.300,179.924,6.053,149.110
C07972=1161.270,8.689,-47.314,179.926,6.053,149.109
C07973=1161.265,8.938,-47.327,179.928,6.054,149.108
C07974=1161.260,9.188,-47.342,179.931,6.055,149.108
C07975=1161.254,9.437,-47.355,179.934,6.055,149.107
C07976=1161.249,9.687,-47.369,179.936,6.056,149.107
C07977=1161.244,9.937,-47.383,179.939,6.057,149.106
C07978=1161.239,10.185,-47.397,179.941,6.058,149.105
C07979=1161.234,10.436,-47.410,179.944,6.059,149.105
C07980=1161.229,10.685,-47.424,179.946,6.059,149.104
C07981=1161.223,10.934,-47.438,179.949,6.060,149.104
C07982=1161.218,11.184,-47.453,179.951,6.061,149.103
C07983=1161.214,11.434,-47.466,179.954,6.061,149.102
C07984=1161.208,11.683,-47.480,179.956,6.063,149.102
C07985=1161.203,11.933,-47.494,179.959,6.063,149.101
C07986=1161.198,12.183,-47.508,179.962,6.064,149.101
C07987=1161.193,12.432,-47.522,179.964,6.065,149.100
C07988=1161.188,12.681,-47.536,179.966,6.065,149.100
C07989=1161.183,12.932,-47.550,179.969,6.066,149.099
C07990=1161.178,13.180,-47.563,179.972,6.067,149.098
C07991=1161.173,13.430,-47.577,179.974,6.068,149.098
C07992=1161.168,13.680,-47.592,179.977,6.068,149.097
C07993=1161.163,13.930,-47.606,179.979,6.069,149.097
C07994=1161.157,14.179,-47.620,179.982,6.070,149.096
C07995=1161.153,14.428,-47.634,179.984,6.071,149.096
C07996=1161.147,14.679,-47.648,179.987,6.072,149.095
C07997=1161.142,14.928,-47.662,179.989,6.073,149.095
C07998=1161.137,15.177,-47.676,179.992,6.073,149.094
C07999=1161.133,15.427,-47.690,179.994,6.074,149.093
C08000=1161.128,15.676,-47.704,179.997,6.074,149.093
C08001=1161.122,15.925,-47.718,179.999,6.075,149.092
C08002=1161.117,16.175,-47.732,-179.998,6.076,149.092
C08003=1161.112,16.425,-47.746,-179.995,6.077,149.091
C08004=1161.107,16.675,-47.761,-179.993,6.078,149.090
C08005=1161.102,16.924,-47.775,-179.991,6.078,149.090
C08006=1161.097,17.173,-47.789,-179.988,6.079,149.089
C08007=1161.092,17.423,-47.803,-179.985,6.080,149.089
C08008=1161.087,17.673,-47.817,-179.983,6.081,149.088
C08009=1161.081,17.922,-47.831,-179.980,6.082,149.087
C08010=1161.076,18.171,-47.846,-179.978,6.082,149.087
C08011=1161.071,18.421,-47.860,-179.975,6.083,149.086
C08012=1161.066,18.671,-47.874,-179.972,6.084,149.086
C08013=1161.061,18.921,-47.888,-179.970,6.085,149.085
C08014=1161.056,19.170,-47.902,-179.967,6.086,149.084
C08015=1161.051,19.419,-47.917,-179.965,6.086,149.084
C08016=1161.046,19.669,-47.931,-179.963,6.087,149.083
C08017=1161.041,19.919,-47.945,-179.960,6.088,149.083
C08018=1161.036,20.168,-47.959,-179.957,6.089,149.082
C08019=1161.030,20.417,-47.973,-179.955,6.090,149.082
C08020=1161.025,20.667,-47.988,-179.952,6.090,149.081
C08021=1161.021,20.916,-48.003,-179.950,6.091,149.081
C08022=1161.016,21.166,-48.017,-179.947,6.092,149.080
C08023=1161.010,21.416,-48.032,-179.945,6.093,149.079
C08024=1161.005,21.666,-48.046,-179.942,6.094,149.079
C08025=1161.000,21.915,-48.060,-179.940,6.094,149.078
C08026=1160.995,22.164,-48.074,-179.937,6.095,149.078
C08027=1160.990,22.414,-48.088,-179.934,6.096,149.077
C08028=1160.985,22.663,-48.103,-179.932,6.097,149.077
C08029=1160.980,22.913,-48.118,-179.929,6.098,149.076
C08030=1160.975,23.163,-48.132,-179.927,6.098,149.075
C08031=1160.970,23.412,-48.146,-179.924,6.100,149.075
C08032=1160.965,23.661,-48.160,-179.922,6.100,149.074
C08033=1160.959,23.911,-48.176,-179.919,6.101,149.074
C08034=1160.954,24.160,-48.190,-179.917,6.102,149.073
C08035=1160.949,24.410,-48.204,-179.914,6.102,149.072
C08036=1160.944,24.660,-48.219,-179.912,6.104,149.072
C08037=1160.940,24.909,-48.234,-179.909,6.104,149.071
C08038=1160.935,25.159,-48.248,-179.907,6.105,149.071
C08039=1160.930,25.408,-48.262,-179.904,6.106,149.070
C08040=1160.924,25.658,-48.277,-179.901,6.107,149.070
C08041=1160.919,25.907,-48.292,-179.899,6.108,149.069
C08042=1160.914,26.156,-48.306,-179.896,6.109,149.069
C08043=1160.909,26.406,-48.320,-179.894,6.109,149.068
C08044=1160.904,26.655,-48.335,-179.891,6.111,149.067
C08045=1160.899,26.905,-48.350,-179.888,6.111,149.067
C08046=1160.894,27.155,-48.364,-179.886,6.112,149.066
C08047=1160.889,27.404,-48.379,-179.884,6.113,149.066
C08048=1160.884,27.674,-48.394,-179.880,6.114,149.065
C08049=1160.878,27.943,-48.411,-179.878,6.115,149.065
C08050=1160.873,28.211,-48.426,-179.875,6.116,149.064
C08051=1160.868,28.480,-48.442,-179.872,6.116,149.063
C08052=1160.862,28.730,-48.457,-179.870,6.117,149.063
C08053=1160.857,28.979,-48.472,-179.867,6.119,149.062
C08054=1160.852,29.229,-48.486,-179.865,6.119,149.062
C08055=1160.847,29.477,-48.501,-179.862,6.120,149.061
C08056=1160.841,29.727,-48.516,-179.860,6.121,149.060
C08057=1160.837,29.977,-48.531,-179.857,6.122,149.060
C08058=1160.832,30.226,-48.545,-179.855,6.123,149.059
C08059=1160.826,30.476,-48.560,-179.852,6.123,149.059
C08060=1160.821,30.725,-48.575,-179.850,6.124,149.058
C08061=1160.816,30.975,-48.589,-179.847,6.125,149.058
C08062=1160.811,31.224,-48.605,-179.844,6.126,149.057
C08063=1160.806,31.474,-48.619,-179.842,6.127,149.056
C08064=1160.801,31.723,-48.634,-179.838,6.128,149.056
C08065=1160.796,31.973,-48.649,-179.836,6.129,149.055
C08066=1160.791,32.222,-48.664,-179.834,6.129,149.055
C08067=1160.786,32.472,-48.678,-179.832,6.130,149.054
C08068=1160.781,32.721,-48.694,-179.828,6.131,149.053
C08069=1160.776,32.971,-48.708,-179.826,6.132,149.053
C08070=1160.771,33.220,-48.723,-179.823,6.133,149.052
C08071=1160.766,33.470,-48.739,-179.821,6.134,149.052
C08072=1160.761,33.720,-48.753,-179.818,6.135,149.051
C08073=1160.757,33.969,-48.768,-179.816,6.136,149.051
C08074=1160.751,34.219,-48.783,-179.813,6.136,149.050
C08075=1160.746,34.468,-48.798,-179.811,6.138,149.050
C08076=1160.741,34.718,-48.814,-179.808,6.138,149.049
C08077=1160.736,34.967,-48.828,-179.806,6.139,149.049
C08078=1160.731,35.217,-48.844,-179.802,6.140,149.048
C08079=1160.726,35.467,-48.858,-179.800,6.141,149.047
C08080=1160.721,35.716,-48.873,-179.798,6.142,149.047
C08081=1160.716,35.965,-48.888,-179.795,6.143,149.046
C08082=1160.711,36.215,-48.903,-179.792,6.144,149.046
C08083=1160.705,36.464,-48.918,-179.790,6.145,149.045
C08084=1160.701,36.713,-48.933,-179.787,6.145,149.044
C08085=1160.695,36.963,-48.948,-179.785,6.147,149.044
C08086=1160.690,37.212,-48.963,-179.782,6.147,149.043
C08087=1160.686,37.462,-48.979,-179.780,6.148,149.043
C08088=1160.681,37.712,-48.993,-179.777,6.149,149.042
C08089=1160.675,37.962,-49.009,-179.775,6.150,149.042
C08090=1160.671,38.211,-49.024,-179.772,6.151,149.041
C08091=1160.665,38.460,-49.040,-179.769,6.152,149.041
C08092=1160.660,38.710,-49.054,-179.766,6.153,149.040
C08093=1160.655,38.959,-49.069,-179.764,6.154,149.040
C08094=1160.650,39.208,-49.084,-179.761,6.155,149.039
C08095=1160.645,39.458,-49.100,-179.759,6.156,149.038
C08096=1160.640,39.708,-49.115,-179.756,6.156,149.038
C08097=1160.635,39.957,-49.130,-179.754,6.158,149.037
C08098=1160.630,40.207,-49.145,-179.751,6.159,149.037
C08099=1160.625,40.456,-49.161,-179.749,6.159,149.036
C08100=1160.620,40.705,-49.176,-179.745,6.161,149.035
C08101=1160.615,40.954,-49.191,-179.743,6.162,149.035
C08102=1160.610,41.205,-49.207,-179.741,6.162,149.034
C08103=1160.605,41.454,-49.222,-179.738,6.164,149.034
C08104=1160.600,41.704,-49.237,-179.735,6.164,149.033
C08105=1160.595,41.953,-49.252,-179.733,6.165,149.033
C08106=1160.590,42.202,-49.268,-179.730,6.167,149.032
C08107=1160.584,42.452,-49.283,-179.728,6.167,149.032
C08108=1160.580,42.701,-49.299,-179.726,6.168,149.031
C08109=1160.575,42.951,-49.314,-179.722,6.169,149.031
C08110=1160.570,43.200,-49.329,-179.720,6.170,149.030
C08111=1160.565,43.450,-49.344,-179.718,6.171,149.029
C08112=1160.559,43.699,-49.360,-179.715,6.172,149.029
C08113=1160.555,43.949,-49.375,-179.712,6.173,149.028
C08114=1160.550,44.198,-49.391,-179.710,6.174,149.028
C08115=1160.544,44.448,-49.406,-179.707,6.175,149.027
C08116=1160.540,44.697,-49.421,-179.705,6.176,149.027
C08117=1160.534,44.946,-49.437,-179.701,6.177,149.026
C08118=1160.530,45.196,-49.453,-179.699,6.178,149.026
C08119=1160.525,45.446,-49.468,-179.697,6.178,149.025
C08120=1160.520,45.695,-49.483,-179.694,6.180,149.025
C08121=1160.514,45.944,-49.499,-179.691,6.181,149.024
C08122=1160.510,46.194,-49.514,-179.689,6.181,149.023
C08123=1160.505,46.444,-49.530,-179.686,6.183,149.023
C08124=1160.499,46.693,-49.545,-179.684,6.184,149.022
C08125=1160.494,46.942,-49.561,-179.680,6.185,149.022
C08126=1160.490,47.192,-49.576,-179.678,6.186,149.021
C08127=1160.485,47.442,-49.592,-179.676,6.186,149.021
C08128=1160.479,47.690,-49.608,-179.673,6.188,149.020
C08129=1160.475,47.940,-49.624,-179.670,6.188,149.019
C08130=1160.470,48.190,-49.639,-179.668,6.189,149.019
C08131=1160.465,48.439,-49.655,-179.665,6.191,149.019
C08132=1160.459,48.688,-49.670,-179.663,6.191,149.018
C08133=1160.454,48.938,-49.686,-179.660,6.193,149.017
C08134=1160.450,49.188,-49.701,-179.657,6.193,149.017
C08135=1160.444,49.437,-49.717,-179.655,6.194,149.016
C08136=1160.440,49.686,-49.734,-179.652,6.196,149.016
C08137=1160.435,49.936,-49.749,-179.650,6.197,149.015
C08138=1160.430,50.185,-49.764,-179.647,6.198,149.015
C08139=1160.425,50.435,-49.780,-179.644,6.199,149.014
C08140=1160.420,50.684,-49.796,-179.642,6.199,149.013
C08141=1160.414,50.934,-49.811,-179.639,6.201,149.013
C08142=1160.410,51.183,-49.828,-179.636,6.201,149.012
C08143=1160.405,51.433,-49.844,-179.634,6.203,149.012
C08144=1160.400,51.682,-49.859,-179.631,6.203,149.011
C08145=1160.395,51.932,-49.875,-179.629,6.204,149.011
C08146=1160.390,52.181,-49.891,-179.626,6.206,149.010
C08147=1160.385,52.430,-49.906,-179.623,6.206,149.010
C08148=1160.380,52.680,-49.922,-179.621,6.208,149.009
C08149=1160.374,52.930,-49.938,-179.618,6.209,149.009
C08150=1160.369,53.178,-49.954,-179.616,6.209,149.008
C08151=1160.365,53.428,-49.970,-179.613,6.211,149.007
C08152=1160.360,53.697,-49.987,-179.611,6.212,149.007
C08153=1160.354,53.965,-50.004,-179.607,6.213,149.006
C08154=1160.349,54.234,-50.021,-179.604,6.214,149.006
C08155=1160.344,54.503,-50.038,-179.602,6.215,149.005
C08156=1160.339,54.752,-50.054,-179.599,6.216,149.005
C08157=1160.334,55.002,-50.070,-179.597,6.217,149.004
C08158=1160.328,55.251,-50.086,-179.593,6.219,149.003
C08159=1160.323,55.500,-50.102,-179.591,6.219,149.003
C08160=1160.319,55.750,-50.118,-179.588,6.220,149.002
C08161=1160.313,55.999,-50.135,-179.586,6.222,149.002
C08162=1160.309,56.249,-50.150,-179.584,6.222,149.001
C08163=1160.303,56.498,-50.166,-179.580,6.224,149.001
C08164=1160.298,56.747,-50.182,-179.578,6.225,149.000
C08165=1160.293,56.997,-50.198,-179.575,6.226,149.000
C08166=1160.288,57.246,-50.215,-179.573,6.227,148.999
C08167=1160.284,57.496,-50.231,-179.570,6.228,148.999
C08168=1160.278,57.745,-50.247,-179.567,6.229,148.998
C08169=1160.274,57.995,-50.263,-179.565,6.229,148.998
C08170=1160.269,58.244,-50.279,-179.562,6.231,148.997
C08171=1160.264,58.494,-50.295,-179.560,6.232,148.997
C08172=1160.259,58.743,-50.311,-179.557,6.233,148.996
C08173=1160.254,58.993,-50.327,-179.555,6.234,148.996
C08174=1160.249,59.241,-50.344,-179.551,6.235,148.995
C08175=1160.243,59.491,-50.359,-179.549,6.236,148.994
C08176=1160.239,59.740,-50.376,-179.546,6.238,148.994
C08177=1160.234,59.990,-50.391,-179.544,6.238,148.993
C08178=1160.229,60.239,-50.408,-179.541,6.240,148.993
C08179=1160.224,60.489,-50.424,-179.538,6.241,148.992
C08180=1160.219,60.738,-50.441,-179.536,6.241,148.992
C08181=1160.213,60.988,-50.457,-179.533,6.243,148.991
C08182=1160.209,61.237,-50.473,-179.531,6.244,148.991
C08183=1160.204,61.486,-50.490,-179.528,6.245,148.990
C08184=1160.199,61.736,-50.506,-179.526,6.246,148.990
C08185=1160.194,61.985,-50.522,-179.522,6.247,148.989
C08186=1160.189,62.234,-50.538,-179.520,6.248,148.988
C08187=1160.184,62.485,-50.554,-179.517,6.250,148.988
C08188=1160.179,62.733,-50.571,-179.515,6.250,148.987
C08189=1160.174,62.983,-50.588,-179.512,6.252,148.987
C08190=1160.169,63.233,-50.604,-179.509,6.252,148.986
C08191=1160.164,63.482,-50.620,-179.507,6.254,148.986
C08192=1160.159,63.731,-50.637,-179.504,6.255,148.985
C08193=1160.154,63.981,-50.653,-179.501,6.256,148.985
C08194=1160.149,64.230,-50.669,-179.499,6.257,148.984
C08195=1160.144,64.480,-50.686,-179.496,6.258,148.984
C08196=1160.139,64.730,-50.702,-179.494,6.259,148.983
C08197=1160.134,64.978,-50.718,-179.491,6.261,148.983
C08198=1160.130,65.228,-50.735,-179.488,6.261,148.982
C08199=1160.125,65.477,-50.751,-179.486,6.263,148.982
C08200=1160.119,65.727,-50.768,-179.483,6.264,148.981
C08201=1160.115,65.977,-50.785,-179.480,6.265,148.981
C08202=1160.110,66.225,-50.801,-179.478,6.266,148.980
C08203=1160.105,66.475,-50.818,-179.475,6.267,148.980
C08204=1160.099,66.724,-50.834,-179.473,6.268,148.979
C08205=1160.095,66.974,-50.850,-179.470,6.270,148.978
C08206=1160.090,67.224,-50.867,-179.467,6.270,148.978
C08207=1160.085,67.472,-50.883,-179.464,6.272,148.977
C08208=1160.080,67.722,-50.901,-179.462,6.273,148.977
C08209=1160.075,67.971,-50.917,-179.459,6.274,148.976
C08210=1160.070,68.220,-50.934,-179.457,6.275,148.976
C08211=1160.066,68.470,-50.950,-179.454,6.276,148.975
C08212=1160.060,68.720,-50.966,-179.451,6.277,148.975
C08213=1160.055,68.969,-50.983,-179.449,6.279,148.974
C08214=1160.051,69.219,-51.000,-179.446,6.279,148.974
C08215=1160.045,69.468,-51.017,-179.443,6.281,148.973
C08216=1160.040,69.717,-51.033,-179.441,6.282,148.973
C08217=1160.036,69.967,-51.050,-179.438,6.283,148.972
C08218=1160.030,70.216,-51.067,-179.436,6.284,148.972
C08219=1160.026,70.465,-51.084,-179.432,6.285,148.971
C08220=1160.021,70.715,-51.100,-179.430,6.286,148.971
C08221=1160.015,70.964,-51.117,-179.428,6.288,148.970
C08222=1160.011,71.213,-51.134,-179.424,6.289,148.969
C08223=1160.006,71.463,-51.150,-179.422,6.290,148.969
C08224=1160.000,71.712,-51.167,-179.419,6.291,148.968
C08225=1159.996,71.961,-51.184,-179.417,6.292,148.968
C08226=1159.991,72.211,-51.201,-179.414,6.294,148.968
C08227=1159.986,72.461,-51.218,-179.411,6.294,148.967
C08228=1159.981,72.709,-51.234,-179.409,6.296,148.966
C08229=1159.976,72.959,-51.252,-179.407,6.297,148.966
C08230=1159.972,73.209,-51.268,-179.403,6.298,148.965
C08231=1159.966,73.458,-51.285,-179.401,6.299,148.965
C08232=1159.961,73.707,-51.302,-179.398,6.300,148.964
C08233=1159.956,73.957,-51.319,-179.395,6.302,148.964
C08234=1159.952,74.207,-51.336,-179.393,6.303,148.963
C08235=1159.947,74.455,-51.353,-179.390,6.304,148.963
C08236=1159.942,74.704,-51.370,-179.388,6.305,148.962
C08237=1159.937,74.954,-51.387,-179.384,6.306,148.962
C08238=1159.932,75.204,-51.404,-179.382,6.307,148.961
C08239=1159.927,75.453,-51.420,-179.380,6.309,148.961
C08240=1159.922,75.702,-51.437,-179.377,6.309,148.960
C08241=1159.917,75.952,-51.454,-179.374,6.311,148.960
C08242=1159.912,76.201,-51.472,-179.371,6.313,148.959
C08243=1159.908,76.450,-51.489,-179.369,6.313,148.959
C08244=1159.902,76.700,-51.506,-179.366,6.315,148.958
C08245=1159.897,76.949,-51.522,-179.363,6.316,148.958
C08246=1159.892,77.199,-51.540,-179.361,6.317,148.957
C08247=1159.888,77.448,-51.557,-179.359,6.318,148.957
C08248=1159.882,77.697,-51.574,-179.355,6.319,148.956
C08249=1159.878,77.946,-51.591,-179.353,6.321,148.956
C08250=1159.872,78.196,-51.608,-179.351,6.322,148.955
C08251=1159.868,78.445,-51.626,-179.347,6.323,148.955
C08252=1159.863,78.695,-51.643,-179.345,6.324,148.954
C08253=1159.858,78.945,-51.660,-179.342,6.326,148.954
C08254=1159.853,79.193,-51.677,-179.339,6.327,148.953
C08255=1159.848,79.442,-51.694,-179.337,6.328,148.953
C08256=1159.842,79.711,-51.713,-179.334,6.329,148.952
C08257=1159.838,79.980,-51.731,-179.331,6.331,148.952
C08258=1159.832,80.248,-51.749,-179.328,6.332,148.951
C08259=1159.827,80.516,-51.769,-179.326,6.333,148.950
C08260=1159.822,80.766,-51.785,-179.323,6.335,148.950
C08261=1159.817,81.016,-51.803,-179.320,6.336,148.949
C08262=1159.812,81.264,-51.820,-179.318,6.337,148.949
C08263=1159.807,81.514,-51.837,-179.314,6.338,148.948
C08264=1159.802,81.763,-51.855,-179.312,6.339,148.948
C08265=1159.797,82.013,-51.872,-179.310,6.341,148.947
C08266=1159.792,82.262,-51.889,-179.306,6.342,148.947
C08267=1159.788,82.511,-51.907,-179.304,6.343,148.946
C08268=1159.782,82.761,-51.924,-179.301,6.345,148.946
C08269=1159.778,83.010,-51.941,-179.299,6.345,148.945
C08270=1159.773,83.260,-51.959,-179.296,6.347,148.945
C08271=1159.767,83.508,-51.976,-179.293,6.348,148.944
C08272=1159.763,83.758,-51.993,-179.291,6.349,148.944
C08273=1159.758,84.007,-52.011,-179.288,6.351,148.943
C08274=1159.753,84.257,-52.028,-179.285,6.352,148.943
C08275=1159.748,84.506,-52.046,-179.283,6.353,148.942
C08276=1159.743,84.755,-52.063,-179.280,6.355,148.942
C08277=1159.738,85.004,-52.081,-179.277,6.355,148.941
C08278=1159.733,85.254,-52.098,-179.275,6.357,148.941
C08279=1159.728,85.503,-52.116,-179.272,6.359,148.940
C08280=1159.724,85.753,-52.133,-179.269,6.359,148.940
C08281=1159.719,86.002,-52.151,-179.266,6.361,148.939
C08282=1159.714,86.251,-52.169,-179.264,6.363,148.939
C08283=1159.709,86.501,-52.186,-179.261,6.363,148.938
C08284=1159.705,86.750,-52.203,-179.258,6.365,148.938
C08285=1159.699,87.000,-52.221,-179.256,6.367,148.937
C08286=1159.695,87.249,-52.239,-179.253,6.367,148.937
C08287=1159.690,87.498,-52.257,-179.250,6.369,148.936
C08288=1159.684,87.748,-52.274,-179.248,6.370,148.936
C08289=1159.679,87.997,-52.292,-179.245,6.371,148.935
C08290=1159.675,88.246,-52.309,-179.242,6.373,148.935
C08291=1159.670,88.496,-52.326,-179.240,6.374,148.934
C08292=1159.665,88.745,-52.344,-179.237,6.375,148.934
C08293=1159.660,88.994,-52.362,-179.234,6.377,148.933
C08294=1159.655,89.244,-52.380,-179.232,6.377,148.933
C08295=1159.650,89.493,-52.398,-179.229,6.379,148.932
C08296=1159.645,89.742,-52.416,-179.226,6.381,148.932
C08297=1159.641,89.992,-52.432,-179.224,6.381,148.931
C08298=1159.636,90.241,-52.450,-179.221,6.383,148.931
C08299=1159.631,90.490,-52.468,-179.218,6.384,148.930
C08300=1159.626,90.739,-52.486,-179.216,6.385,148.930
C08301=1159.621,90.988,-52.504,-179.213,6.387,148.930
C08302=1159.616,91.238,-52.521,-179.210,6.388,148.929
C08303=1159.611,91.487,-52.539,-179.208,6.389,148.928
C08304=1159.606,91.737,-52.557,-179.205,6.391,148.928
C08305=1159.601,91.986,-52.575,-179.202,6.392,148.927
C08306=1159.596,92.235,-52.593,-179.200,6.393,148.927
C08307=1159.591,92.485,-52.611,-179.197,6.395,148.927
C08308=1159.586,92.734,-52.629,-179.194,6.396,148.926
C08309=1159.581,92.983,-52.647,-179.191,6.398,148.925
C08310=1159.576,93.232,-52.665,-179.189,6.399,148.925
C08311=1159.571,93.481,-52.683,-179.186,6.400,148.925
C08312=1159.567,93.731,-52.701,-179.183,6.402,148.924
C08313=1159.562,93.980,-52.719,-179.181,6.403,148.924
C08314=1159.557,94.230,-52.737,-179.178,6.404,148.923
C08315=1159.552,94.479,-52.754,-179.175,6.406,148.923
C08316=1159.547,94.729,-52.772,-179.173,6.407,148.922
C08317=1159.542,94.978,-52.790,-179.170,6.408,148.922
C08318=1159.537,95.227,-52.808,-179.167,6.410,148.921
C08319=1159.532,95.476,-52.826,-179.165,6.410,148.921
C08320=1159.527,95.725,-52.844,-179.162,6.412,148.920
C08321=1159.523,95.975,-52.862,-179.159,6.414,148.920
C08322=1159.518,96.224,-52.880,-179.156,6.415,148.919
C08323=1159.513,96.473,-52.898,-179.154,6.416,148.919
C08324=1159.508,96.723,-52.916,-179.151,6.418,148.918
C08325=1159.503,96.972,-52.934,-179.148,6.419,148.918
C08326=1159.499,97.221,-52.952,-179.146,6.420,148.917
C08327=1159.494,97.471,-52.971,-179.143,6.422,148.917
C08328=1159.489,97.720,-52.989,-179.140,6.423,148.916
C08329=1159.484,97.969,-53.007,-179.137,6.425,148.916
C08330=1159.479,98.219,-53.025,-179.135,6.426,148.915
C08331=1159.474,98.467,-53.044,-179.132,6.427,148.915
C08332=1159.469,98.716,-53.062,-179.130,6.429,148.915
C08333=1159.465,98.966,-53.080,-179.126,6.430,148.914
C08334=1159.460,99.216,-53.098,-179.124,6.431,148.913
C08335=1159.455,99.465,-53.116,-179.121,6.433,148.913
C08336=1159.450,99.714,-53.134,-179.119,6.435,148.913
C08337=1159.445,99.963,-53.153,-179.116,6.435,148.912
C08338=1159.440,100.213,-53.171,-179.113,6.437,148.912
C08339=1159.436,100.462,-53.190,-179.111,6.439,148.911
C08340=1159.431,100.711,-53.208,-179.107,6.440,148.911
C08341=1159.426,100.960,-53.226,-179.105,6.441,148.910
C08342=1159.422,101.210,-53.244,-179.103,6.442,148.910
C08343=1159.416,101.460,-53.263,-179.100,6.444,148.909
C08344=1159.411,101.708,-53.281,-179.097,6.446,148.909
C08345=1159.406,101.957,-53.299,-179.095,6.446,148.908
C08346=1159.401,102.206,-53.317,-179.092,6.448,148.908
C08347=1159.396,102.457,-53.336,-179.089,6.450,148.907
C08348=1159.391,102.706,-53.354,-179.086,6.451,148.907
C08349=1159.387,102.954,-53.373,-179.084,6.452,148.906
C08350=1159.383,103.204,-53.391,-179.081,6.454,148.906
C08351=1159.377,103.454,-53.410,-179.078,6.455,148.906
C08352=1159.372,103.702,-53.428,-179.075,6.457,148.905
C08353=1159.367,103.951,-53.446,-179.073,6.458,148.904
C08354=1159.363,104.201,-53.465,-179.070,6.459,148.904
C08355=1159.358,104.450,-53.484,-179.068,6.461,148.904
C08356=1159.353,104.699,-53.502,-179.064,6.462,148.903
C08357=1159.349,104.949,-53.520,-179.062,6.464,148.903
C08358=1159.343,105.198,-53.540,-179.059,6.465,148.902
C08359=1159.338,105.447,-53.558,-179.057,6.467,148.902
C08360=1159.332,105.716,-53.578,-179.054,6.468,148.901
C08361=1159.328,105.984,-53.598,-179.051,6.470,148.901
C08362=1159.322,106.253,-53.618,-179.048,6.471,148.900
C08363=1159.317,106.521,-53.638,-179.045,6.473,148.900
C08364=1159.313,106.770,-53.656,-179.042,6.475,148.899
C08365=1159.308,107.020,-53.675,-179.039,6.476,148.899
C08366=1159.303,107.268,-53.694,-179.037,6.477,148.898
C08367=1159.297,107.518,-53.713,-179.034,6.478,148.898
C08368=1159.293,107.768,-53.731,-179.031,6.480,148.897
C08369=1159.289,108.016,-53.750,-179.029,6.482,148.897
C08370=1159.283,108.266,-53.768,-179.026,6.484,148.897
C08371=1159.279,108.515,-53.787,-179.023,6.484,148.896
C08372=1159.273,108.764,-53.806,-179.021,6.486,148.896
C08373=1159.269,109.014,-53.825,-179.018,6.488,148.895
C08374=1159.265,109.262,-53.844,-179.015,6.489,148.895
C08375=1159.259,109.512,-53.862,-179.012,6.491,148.894
C08376=1159.255,109.761,-53.881,-179.010,6.491,148.894
C08377=1159.249,110.010,-53.900,-179.007,6.493,148.893
C08378=1159.245,110.260,-53.919,-179.004,6.495,148.893
C08379=1159.240,110.509,-53.937,-179.002,6.497,148.892
C08380=1159.235,110.758,-53.956,-178.998,6.498,148.892
C08381=1159.230,111.007,-53.976,-178.996,6.499,148.891
C08382=1159.225,111.257,-53.994,-178.994,6.501,148.891
C08383=1159.221,111.506,-54.013,-178.991,6.502,148.891
C08384=1159.216,111.755,-54.031,-178.988,6.504,148.890
C08385=1159.211,112.005,-54.051,-178.985,6.505,148.890
C08386=1159.206,112.253,-54.070,-178.982,6.507,148.889
C08387=1159.201,112.503,-54.088,-178.980,6.508,148.889
C08388=1159.197,112.752,-54.107,-178.977,6.510,148.888
C08389=1159.191,113.001,-54.127,-178.975,6.511,148.888
C08390=1159.187,113.251,-54.145,-178.971,6.513,148.887
C08391=1159.182,113.500,-54.164,-178.969,6.514,148.887
C08392=1159.177,113.749,-54.184,-178.966,6.516,148.887
C08393=1159.172,113.998,-54.203,-178.964,6.517,148.886
C08394=1159.167,114.248,-54.222,-178.961,6.519,148.886
C08395=1159.163,114.497,-54.240,-178.958,6.520,148.885
C08396=1159.158,114.746,-54.260,-178.955,6.522,148.885
C08397=1159.153,114.995,-54.279,-178.953,6.523,148.884
C08398=1159.148,115.245,-54.298,-178.950,6.525,148.884
C08399=1159.143,115.494,-54.317,-178.948,6.526,148.883
C08400=1159.139,115.743,-54.336,-178.945,6.527,148.883
C08401=1159.134,115.992,-54.355,-178.942,6.529,148.882
C08402=1159.129,116.241,-54.375,-178.939,6.531,148.882
C08403=1159.124,116.490,-54.394,-178.936,6.533,148.882
C08404=1159.119,116.740,-54.412,-178.934,6.534,148.881
C08405=1159.114,116.989,-54.432,-178.931,6.536,148.881
C08406=1159.110,117.238,-54.451,-178.928,6.537,148.880
C08407=1159.105,117.487,-54.470,-178.926,6.538,148.880
C08408=1159.100,117.737,-54.490,-178.923,6.540,148.879
C08409=1159.095,117.985,-54.508,-178.920,6.542,148.879
C08410=1159.090,118.235,-54.528,-178.917,6.543,148.879
C08411=1159.085,118.484,-54.547,-178.915,6.545,148.878
C08412=1159.081,118.733,-54.566,-178.912,6.546,148.878
C08413=1159.076,118.983,-54.586,-178.909,6.547,148.877
C08414=1159.071,119.232,-54.605,-178.907,6.549,148.877
C08415=1159.066,119.482,-54.624,-178.904,6.551,148.876
C08416=1159.061,119.730,-54.643,-178.901,6.552,148.876
C08417=1159.057,119.980,-54.663,-178.899,6.554,148.876
C08418=1159.051,120.229,-54.682,-178.895,6.556,148.875
C08419=1159.047,120.478,-54.702,-178.893,6.557,148.875
C08420=1159.043,120.727,-54.721,-178.890,6.559,148.874
C08421=1159.037,120.976,-54.740,-178.888,6.560,148.874
C08422=1159.033,121.225,-54.760,-178.885,6.562,148.873
C08423=1159.027,121.474,-54.780,-178.882,6.563,148.873
C08424=1159.023,121.724,-54.799,-178.880,6.565,148.872
C08425=1159.019,121.973,-54.818,-178.876,6.566,148.872
C08426=1159.013,122.222,-54.838,-178.874,6.568,148.871
C08427=1159.009,122.471,-54.857,-178.871,6.570,148.871
C08428=1159.004,122.721,-54.877,-178.868,6.571,148.871
C08429=1158.998,122.970,-54.896,-178.866,6.573,148.870
C08430=1158.994,123.219,-54.915,-178.863,6.575,148.870
C08431=1158.990,123.469,-54.935,-178.861,6.576,148.869
C08432=1158.985,123.717,-54.955,-178.858,6.577,148.869
C08433=1158.980,123.966,-54.975,-178.855,6.579,148.868
C08434=1158.975,124.216,-54.994,-178.852,6.581,148.868
C08435=1158.970,124.465,-55.014,-178.849,6.582,148.868
C08436=1158.965,124.715,-55.033,-178.847,6.584,148.867
C08437=1158.960,124.964,-55.053,-178.844,6.586,148.867
C08438=1158.956,125.212,-55.072,-178.841,6.587,148.866
C08439=1158.951,125.462,-55.092,-178.839,6.589,148.866
C08440=1158.947,125.711,-55.112,-178.835,6.591,148.865
C08441=1158.941,125.960,-55.131,-178.833,6.592,148.865
C08442=1158.937,126.209,-55.151,-178.831,6.593,148.865
C08443=1158.932,126.459,-55.171,-178.828,6.595,148.864
C08444=1158.927,126.707,-55.190,-178.825,6.597,148.864
C08445=1158.922,126.956,-55.211,-178.822,6.598,148.863
C08446=1158.918,127.206,-55.230,-178.820,6.600,148.863
C08447=1158.913,127.455,-55.250,-178.817,6.602,148.863
C08448=1158.907,127.704,-55.269,-178.814,6.603,148.862
C08449=1158.903,127.953,-55.290,-178.811,6.605,148.862
C08450=1158.898,128.203,-55.309,-178.808,6.607,148.861
C08451=1158.894,128.452,-55.330,-178.806,6.608,148.861
C08452=1158.889,128.701,-55.349,-178.803,6.610,148.860
C08453=1158.884,128.950,-55.369,-178.800,6.612,148.860
C08454=1158.879,129.199,-55.389,-178.797,6.613,148.860
C08455=1158.875,129.449,-55.409,-178.795,6.615,148.859
C08456=1158.869,129.698,-55.428,-178.792,6.617,148.859
C08457=1158.865,129.947,-55.448,-178.789,6.619,148.858
C08458=1158.860,130.196,-55.468,-178.787,6.620,148.858
C08459=1158.856,130.445,-55.488,-178.784,6.621,148.857
C08460=1158.851,130.695,-55.508,-178.781,6.623,148.857
C08461=1158.846,130.943,-55.528,-178.779,6.624,148.857
C08462=1158.841,131.192,-55.548,-178.776,6.626,148.856
C08463=1158.837,131.441,-55.568,-178.773,6.628,148.856
C08464=1158.831,131.710,-55.590,-178.770,6.629,148.855
C08465=1158.826,131.979,-55.611,-178.767,6.632,148.855
C08466=1158.821,132.247,-55.633,-178.764,6.633,148.854
C08467=1158.816,132.516,-55.654,-178.761,6.635,148.854
C08468=1158.811,132.765,-55.675,-178.759,6.637,148.854
C08469=1158.807,133.015,-55.694,-178.756,6.639,148.853
C08470=1158.801,133.263,-55.715,-178.753,6.640,148.853
C08471=1158.796,133.513,-55.735,-178.750,6.642,148.853
C08472=1158.792,133.762,-55.755,-178.748,6.644,148.852
C08473=1158.787,134.011,-55.775,-178.745,6.645,148.852
C08474=1158.783,134.260,-55.795,-178.742,6.647,148.851
C08475=1158.778,134.509,-55.815,-178.740,6.649,148.851
C08476=1158.772,134.758,-55.835,-178.737,6.651,148.851
C08477=1158.768,135.007,-55.856,-178.734,6.652,148.850
C08478=1158.763,135.256,-55.876,-178.731,6.654,148.850
C08479=1158.758,135.506,-55.896,-178.728,6.655,148.849
C08480=1158.754,135.755,-55.916,-178.726,6.657,148.849
C08481=1158.749,136.004,-55.937,-178.723,6.659,148.848
C08482=1158.744,136.254,-55.957,-178.720,6.661,148.848
C08483=1158.740,136.502,-55.977,-178.717,6.662,148.848
C08484=1158.735,136.751,-55.997,-178.715,6.664,148.847
C08485=1158.729,137.000,-56.018,-178.712,6.666,148.847
C08486=1158.725,137.250,-56.038,-178.709,6.667,148.846
C08487=1158.720,137.498,-56.058,-178.707,6.669,148.846
C08488=1158.716,137.747,-56.078,-178.704,6.671,148.846
C08489=1158.711,137.997,-56.099,-178.701,6.673,148.845
C08490=1158.706,138.246,-56.119,-178.699,6.674,148.845
C08491=1158.701,138.495,-56.139,-178.696,6.676,148.844
C08492=1158.696,138.744,-56.160,-178.693,6.678,148.844
C08493=1158.692,138.993,-56.181,-178.690,6.680,148.844
C08494=1158.687,139.242,-56.201,-178.688,6.681,148.843
C08495=1158.682,139.492,-56.221,-178.685,6.683,148.843
C08496=1158.677,139.741,-56.242,-178.682,6.685,148.843
C08497=1158.673,139.990,-56.262,-178.680,6.686,148.842
C08498=1158.668,140.239,-56.283,-178.677,6.688,148.842
C08499=1158.663,140.488,-56.303,-178.674,6.690,148.841
C08500=1158.659,140.737,-56.324,-178.671,6.692,148.841
C08501=1158.654,140.987,-56.345,-178.668,6.693,148.840
C08502=1158.649,141.236,-56.365,-178.666,6.695,148.840
C08503=1158.645,141.484,-56.385,-178.663,6.696,148.840
C08504=1158.640,141.734,-56.406,-178.660,6.698,148.839
C08505=1158.635,141.983,-56.427,-178.657,6.700,148.839
C08506=1158.630,142.232,-56.448,-178.655,6.702,148.838
C08507=1158.626,142.481,-56.468,-178.652,6.703,148.838
C08508=1158.621,142.730,-56.488,-178.649,6.705,148.838
C08509=1158.616,142.979,-56.509,-178.647,6.707,148.837
C08510=1158.612,143.228,-56.530,-178.643,6.709,148.837
C08511=1158.606,143.477,-56.551,-178.641,6.711,148.837
C08512=1158.602,143.726,-56.571,-178.638,6.713,148.836
C08513=1158.597,143.975,-56.592,-178.635,6.715,148.836
C08514=1158.592,144.224,-56.613,-178.633,6.716,148.835
C08515=1158.587,144.474,-56.633,-178.630,6.718,148.835
C08516=1158.583,144.723,-56.654,-178.627,6.720,148.835
C08517=1158.578,144.972,-56.675,-178.624,6.721,148.834
C08518=1158.573,145.221,-56.695,-178.622,6.723,148.834
C08519=1158.568,145.470,-56.716,-178.619,6.725,148.833
C08520=1158.564,145.720,-56.737,-178.616,6.727,148.833
C08521=1158.559,145.969,-56.758,-178.614,6.728,148.833
C08522=1158.555,146.217,-56.779,-178.611,6.730,148.832
C08523=1158.550,146.467,-56.800,-178.608,6.732,148.832
C08524=1158.545,146.716,-56.820,-178.605,6.734,148.832
C08525=1158.540,146.965,-56.841,-178.603,6.735,148.831
C08526=1158.536,147.214,-56.862,-178.599,6.738,148.831
C08527=1158.530,147.463,-56.883,-178.597,6.740,148.831
C08528=1158.526,147.712,-56.904,-178.595,6.742,148.830
C08529=1158.521,147.961,-56.925,-178.592,6.743,148.830
C08530=1158.517,148.211,-56.946,-178.589,6.745,148.829
C08531=1158.512,148.460,-56.966,-178.586,6.747,148.829
C08532=1158.507,148.708,-56.988,-178.584,6.749,148.829
C08533=1158.502,148.957,-57.009,-178.581,6.750,148.828
C08534=1158.498,149.206,-57.029,-178.578,6.752,148.828
C08535=1158.493,149.455,-57.051,-178.576,6.754,148.828
C08536=1158.488,149.704,-57.071,-178.573,6.756,148.827
C08537=1158.484,149.954,-57.093,-178.570,6.758,148.827
C08538=1158.479,150.203,-57.114,-178.567,6.760,148.826
C08539=1158.474,150.452,-57.135,-178.564,6.762,148.826
C08540=1158.469,150.701,-57.156,-178.562,6.763,148.826
C08541=1158.464,150.949,-57.177,-178.559,6.765,148.825
C08542=1158.460,151.198,-57.198,-178.556,6.767,148.825
C08543=1158.455,151.448,-57.219,-178.553,6.768,148.825
C08544=1158.451,151.697,-57.241,-178.551,6.770,148.824
C08545=1158.445,151.946,-57.262,-178.548,6.772,148.824
C08546=1158.441,152.195,-57.282,-178.545,6.774,148.823
C08547=1158.436,152.444,-57.304,-178.542,6.776,148.823
C08548=1158.432,152.694,-57.325,-178.539,6.778,148.823
C08549=1158.427,152.942,-57.347,-178.537,6.780,148.822
C08550=1158.422,153.191,-57.367,-178.534,6.782,148.822
C08551=1158.417,153.440,-57.389,-178.532,6.783,148.822
C08552=1158.413,153.690,-57.410,-178.529,6.785,148.821
C08553=1158.408,153.939,-57.432,-178.526,6.787,148.821
C08554=1158.403,154.188,-57.452,-178.524,6.789,148.821
C08555=1158.399,154.436,-57.474,-178.520,6.791,148.820
C08556=1158.394,154.686,-57.495,-178.518,6.793,148.820
C08557=1158.389,154.935,-57.517,-178.515,6.795,148.819
C08558=1158.384,155.184,-57.538,-178.512,6.796,148.819
C08559=1158.380,155.432,-57.559,-178.510,6.798,148.819
C08560=1158.376,155.682,-57.581,-178.507,6.800,148.818
C08561=1158.370,155.931,-57.602,-178.504,6.802,148.818
C08562=1158.366,156.180,-57.624,-178.501,6.804,148.818
C08563=1158.360,156.429,-57.645,-178.499,6.806,148.817
C08564=1158.356,156.678,-57.667,-178.496,6.808,148.817
C08565=1158.352,156.927,-57.688,-178.493,6.810,148.817
C08566=1158.347,157.176,-57.709,-178.491,6.812,148.816
C08567=1158.343,157.425,-57.731,-178.488,6.813,148.816
C08568=1158.337,157.695,-57.754,-178.485,6.816,148.816
C08569=1158.332,157.964,-57.777,-178.482,6.818,148.815
C08570=1158.326,158.232,-57.801,-178.479,6.820,148.815
C08571=1158.322,158.501,-57.823,-178.476,6.822,148.814
C08572=1158.317,158.750,-57.846,-178.473,6.824,148.814
C08573=1158.313,158.999,-57.867,-178.470,6.825,148.814
C08574=1158.307,159.248,-57.888,-178.468,6.827,148.813
C08575=1158.303,159.497,-57.910,-178.464,6.830,148.813
C08576=1158.298,159.746,-57.932,-178.462,6.831,148.813
C08577=1158.293,159.995,-57.954,-178.459,6.833,148.812
C08578=1158.289,160.244,-57.975,-178.456,6.835,148.812
C08579=1158.284,160.493,-57.997,-178.454,6.837,148.812
C08580=1158.280,160.742,-58.019,-178.451,6.839,148.811
C08581=1158.275,160.991,-58.040,-178.448,6.841,148.811
C08582=1158.270,161.240,-58.062,-178.446,6.843,148.811
C08583=1158.265,161.490,-58.083,-178.443,6.845,148.810
C08584=1158.261,161.738,-58.105,-178.440,6.846,148.810
C08585=1158.256,161.988,-58.127,-178.437,6.848,148.809
C08586=1158.251,162.236,-58.149,-178.434,6.851,148.809
C08587=1158.247,162.485,-58.170,-178.432,6.853,148.809
C08588=1158.242,162.734,-58.192,-178.429,6.855,148.809
C08589=1158.237,162.983,-58.214,-178.427,6.856,148.808
C08590=1158.233,163.232,-58.236,-178.424,6.858,148.808
C08591=1158.228,163.481,-58.258,-178.421,6.861,148.807
C08592=1158.224,163.730,-58.280,-178.418,6.862,148.807
C08593=1158.219,163.979,-58.302,-178.415,6.864,148.807
C08594=1158.214,164.228,-58.323,-178.413,6.866,148.807
C08595=1158.210,164.477,-58.345,-178.410,6.868,148.806
C08596=1158.205,164.726,-58.367,-178.407,6.870,148.806
C08597=1158.200,164.975,-58.390,-178.404,6.872,148.805
C08598=1158.195,165.224,-58.411,-178.402,6.874,148.805
C08599=1158.191,165.473,-58.433,-178.399,6.876,148.805
C08600=1158.186,165.722,-58.455,-178.397,6.878,148.805
C08601=1158.182,165.971,-58.477,-178.393,6.880,148.804
C08602=1158.177,166.220,-58.499,-178.391,6.882,148.804
C08603=1158.173,166.469,-58.521,-178.388,6.884,148.803
C08604=1158.167,166.718,-58.543,-178.385,6.886,148.803
C08605=1158.163,166.967,-58.565,-178.382,6.888,148.803
C08606=1158.158,167.216,-58.587,-178.379,6.890,148.802
C08607=1158.154,167.465,-58.609,-178.377,6.892,148.802
C08608=1158.149,167.714,-58.631,-178.374,6.894,148.802
C08609=1158.144,167.963,-58.654,-178.372,6.895,148.802
C08610=1158.139,168.212,-58.676,-178.368,6.898,148.801
C08611=1158.135,168.461,-58.698,-178.366,6.900,148.801
C08612=1158.130,168.710,-58.719,-178.364,6.902,148.801
C08613=1158.125,168.959,-58.742,-178.361,6.904,148.800
C08614=1158.120,169.208,-58.764,-178.358,6.906,148.800
C08615=1158.116,169.457,-58.786,-178.355,6.908,148.800
C08616=1158.111,169.705,-58.808,-178.352,6.910,148.799
C08617=1158.106,169.955,-58.831,-178.349,6.911,148.799
C08618=1158.102,170.204,-58.853,-178.347,6.914,148.799
C08619=1158.098,170.452,-58.875,-178.344,6.916,148.798
C08620=1158.093,170.702,-58.897,-178.341,6.918,148.798
C08621=1158.088,170.951,-58.920,-178.339,6.920,148.798
C08622=1158.084,171.199,-58.942,-178.335,6.922,148.797
C08623=1158.079,171.448,-58.964,-178.333,6.924,148.797
C08624=1158.074,171.698,-58.987,-178.330,6.926,148.797
C08625=1158.070,171.947,-59.009,-178.328,6.928,148.796
C08626=1158.065,172.195,-59.031,-178.324,6.930,148.796
C08627=1158.060,172.445,-59.054,-178.322,6.932,148.796
C08628=1158.056,172.693,-59.077,-178.320,6.934,148.795
C08629=1158.051,172.942,-59.098,-178.316,6.937,148.795
C08630=1158.046,173.192,-59.121,-178.314,6.938,148.795
C08631=1158.042,173.440,-59.143,-178.311,6.940,148.794
C08632=1158.037,173.689,-59.166,-178.309,6.942,148.794
C08633=1158.033,173.938,-59.189,-178.305,6.945,148.794
C08634=1158.028,174.187,-59.210,-178.303,6.947,148.794
C08635=1158.023,174.436,-59.233,-178.300,6.948,148.793
C08636=1158.019,174.685,-59.256,-178.298,6.950,148.793
C08637=1158.013,174.934,-59.278,-178.295,6.953,148.793
C08638=1158.009,175.183,-59.301,-178.292,6.955,148.792
C08639=1158.004,175.432,-59.323,-178.289,6.956,148.792
C08640=1158.000,175.680,-59.346,-178.286,6.959,148.792
C08641=1157.995,175.930,-59.368,-178.284,6.961,148.791
C08642=1157.991,176.179,-59.391,-178.281,6.963,148.791
C08643=1157.986,176.427,-59.414,-178.278,6.965,148.791
C08644=1157.981,176.676,-59.436,-178.275,6.967,148.790
C08645=1157.977,176.925,-59.459,-178.273,6.969,148.790
C08646=1157.972,177.174,-59.481,-178.270,6.971,148.790
C08647=1157.968,177.423,-59.504,-178.267,6.974,148.790
C08648=1157.963,177.673,-59.527,-178.264,6.975,148.789
C08649=1157.959,177.921,-59.549,-178.262,6.977,148.789
C08650=1157.953,178.170,-59.572,-178.259,6.980,148.789
C08651=1157.948,178.419,-59.595,-178.256,6.982,148.788
C08652=1157.944,178.668,-59.618,-178.253,6.983,148.788
C08653=1157.940,178.917,-59.641,-178.250,6.986,148.788
C08654=1157.935,179.166,-59.663,-178.248,6.988,148.787
C08655=1157.930,179.415,-59.686,-178.245,6.990,148.787
C08656=1157.926,179.663,-59.709,-178.243,6.992,148.787
C08657=1157.921,179.913,-59.732,-178.240,6.995,148.787
C08658=1157.917,180.161,-59.754,-178.237,6.996,148.786
C08659=1157.912,180.410,-59.777,-178.234,6.998,148.786
C08660=1157.907,180.659,-59.801,-178.231,7.001,148.786
C08661=1157.903,180.908,-59.823,-178.229,7.003,148.785
C08662=1157.898,181.157,-59.846,-178.226,7.004,148.785
C08663=1157.893,181.406,-59.869,-178.223,7.007,148.785
C08664=1157.889,181.655,-59.892,-178.221,7.009,148.785
C08665=1157.884,181.904,-59.915,-178.218,7.011,148.784
C08666=1157.880,182.153,-59.937,-178.215,7.013,148.784
C08667=1157.875,182.401,-59.960,-178.212,7.016,148.784
C08668=1157.870,182.650,-59.984,-178.210,7.017,148.783
C08669=1157.866,182.899,-60.007,-178.206,7.020,148.783
C08670=1157.861,183.148,-60.030,-178.204,7.022,148.783
C08671=1157.857,183.397,-60.053,-178.201,7.025,148.783
C08672=1157.851,183.667,-60.078,-178.198,7.026,148.782
C08673=1157.847,183.936,-60.103,-178.195,7.029,148.782
C08674=1157.841,184.206,-60.128,-178.192,7.031,148.782
C08675=1157.836,184.476,-60.153,-178.189,7.033,148.781
C08676=1157.832,184.725,-60.176,-178.187,7.035,148.781
C08677=1157.827,184.974,-60.199,-178.184,7.038,148.781
C08678=1157.823,185.223,-60.222,-178.181,7.040,148.780
C08679=1157.818,185.472,-60.246,-178.179,7.042,148.780
C08680=1157.813,185.720,-60.268,-178.175,7.044,148.780
C08681=1157.809,185.969,-60.291,-178.173,7.046,148.780
C08682=1157.804,186.218,-60.315,-178.170,7.049,148.779
C08683=1157.799,186.467,-60.338,-178.167,7.051,148.779
C08684=1157.795,186.716,-60.361,-178.165,7.052,148.779
C08685=1157.791,186.965,-60.384,-178.162,7.055,148.779
C08686=1157.786,187.214,-60.408,-178.159,7.057,148.778
C08687=1157.781,187.463,-60.431,-178.156,7.059,148.778
C08688=1157.777,187.711,-60.455,-178.154,7.062,148.778
C08689=1157.772,187.960,-60.478,-178.151,7.064,148.777
C08690=1157.767,188.208,-60.501,-178.148,7.066,148.777
C08691=1157.763,188.457,-60.524,-178.145,7.068,148.777
C08692=1157.758,188.706,-60.547,-178.143,7.070,148.777
C08693=1157.754,188.955,-60.571,-178.140,7.073,148.776
C08694=1157.749,189.204,-60.594,-178.137,7.075,148.776
C08695=1157.744,189.453,-60.618,-178.134,7.077,148.776
C08696=1157.740,189.702,-60.642,-178.131,7.079,148.775
C08697=1157.735,189.951,-60.665,-178.129,7.081,148.775
C08698=1157.730,190.200,-60.688,-178.126,7.084,148.775
C08699=1157.726,190.449,-60.712,-178.124,7.086,148.775
C08700=1157.721,190.697,-60.736,-178.120,7.088,148.774
C08701=1157.717,190.946,-60.759,-178.118,7.090,148.774
C08702=1157.712,191.195,-60.782,-178.116,7.092,148.774
C08703=1157.707,191.444,-60.806,-178.112,7.095,148.774
C08704=1157.703,191.693,-60.830,-178.110,7.097,148.773
C08705=1157.699,191.941,-60.853,-178.107,7.099,148.773
C08706=1157.694,192.190,-60.876,-178.104,7.101,148.773
C08707=1157.690,192.439,-60.900,-178.102,7.103,148.773
C08708=1157.685,192.688,-60.923,-178.099,7.106,148.772
C08709=1157.680,192.937,-60.947,-178.096,7.108,148.772
C08710=1157.675,193.186,-60.972,-178.093,7.111,148.772
C08711=1157.670,193.435,-60.995,-178.090,7.112,148.772
C08712=1157.666,193.684,-61.018,-178.088,7.114,148.771
C08713=1157.661,193.932,-61.042,-178.085,7.117,148.771
C08714=1157.657,194.181,-61.066,-178.082,7.119,148.771
C08715=1157.652,194.430,-61.089,-178.080,7.122,148.771
C08716=1157.648,194.679,-61.113,-178.077,7.123,148.770
C08717=1157.643,194.928,-61.136,-178.074,7.126,148.770
C08718=1157.638,195.176,-61.161,-178.071,7.128,148.770
C08719=1157.634,195.426,-61.184,-178.068,7.131,148.769
C08720=1157.630,195.674,-61.208,-178.066,7.133,148.769
C08721=1157.625,195.923,-61.232,-178.063,7.135,148.769
C08722=1157.621,196.172,-61.256,-178.060,7.137,148.769
C08723=1157.616,196.421,-61.279,-178.058,7.139,148.769
C08724=1157.611,196.669,-61.304,-178.054,7.142,148.768
C08725=1157.606,196.918,-61.327,-178.052,7.144,148.768
C08726=1157.602,197.167,-61.351,-178.049,7.146,148.768
C08727=1157.597,197.416,-61.375,-178.047,7.149,148.768
C08728=1157.593,197.664,-61.399,-178.044,7.151,148.767
C08729=1157.589,197.913,-61.423,-178.041,7.153,148.767
C08730=1157.584,198.163,-61.447,-178.039,7.155,148.767
C08731=1157.579,198.411,-61.471,-178.035,7.158,148.766
C08732=1157.575,198.660,-61.494,-178.033,7.160,148.766
C08733=1157.570,198.909,-61.519,-178.030,7.162,148.766
C08734=1157.566,199.157,-61.543,-178.028,7.164,148.766
C08735=1157.560,199.406,-61.567,-178.024,7.167,148.766
C08736=1157.557,199.655,-61.591,-178.022,7.169,148.765
C08737=1157.552,199.904,-61.615,-178.019,7.172,148.765
C08738=1157.547,200.153,-61.638,-178.016,7.173,148.765
C08739=1157.543,200.401,-61.663,-178.014,7.176,148.765
C08740=1157.538,200.650,-61.687,-178.011,7.178,148.764
C08741=1157.534,200.899,-61.712,-178.008,7.181,148.764
C08742=1157.529,201.148,-61.735,-178.005,7.183,148.764
C08743=1157.524,201.397,-61.760,-178.003,7.186,148.764
C08744=1157.520,201.645,-61.784,-178.000,7.187,148.763
C08745=1157.516,201.894,-61.808,-177.997,7.190,148.763
C08746=1157.511,202.143,-61.832,-177.994,7.192,148.763
C08747=1157.506,202.392,-61.856,-177.991,7.195,148.763
C08748=1157.502,202.641,-61.880,-177.989,7.197,148.762
C08749=1157.497,202.889,-61.904,-177.986,7.199,148.762
C08750=1157.493,203.138,-61.929,-177.983,7.202,148.762
C08751=1157.489,203.387,-61.953,-177.980,7.204,148.762
C08752=1157.484,203.636,-61.977,-177.978,7.206,148.762
C08753=1157.479,203.885,-62.001,-177.975,7.208,148.761
C08754=1157.475,204.134,-62.026,-177.973,7.211,148.761
C08755=1157.470,204.382,-62.051,-177.969,7.214,148.761
C08756=1157.465,204.631,-62.075,-177.967,7.216,148.761
C08757=1157.461,204.879,-62.099,-177.964,7.218,148.760
C08758=1157.456,205.129,-62.124,-177.962,7.220,148.760
C08759=1157.452,205.377,-62.148,-177.958,7.223,148.760
C08760=1157.447,205.626,-62.173,-177.956,7.225,148.760
C08761=1157.443,205.874,-62.197,-177.953,7.228,148.759
C08762=1157.439,206.123,-62.221,-177.951,7.230,148.759
C08763=1157.434,206.372,-62.246,-177.947,7.232,148.759
C08764=1157.429,206.620,-62.270,-177.945,7.234,148.759
C08765=1157.425,206.870,-62.295,-177.942,7.237,148.759
C08766=1157.420,207.118,-62.319,-177.940,7.239,148.758
C08767=1157.415,207.367,-62.344,-177.937,7.242,148.758
C08768=1157.411,207.616,-62.368,-177.934,7.244,148.758
C08769=1157.406,207.865,-62.393,-177.931,7.246,148.758
C08770=1157.402,208.113,-62.417,-177.929,7.248,148.758
C08771=1157.397,208.363,-62.442,-177.926,7.251,148.757
C08772=1157.393,208.611,-62.466,-177.923,7.253,148.757
C08773=1157.388,208.859,-62.491,-177.920,7.256,148.757
C08774=1157.384,209.108,-62.516,-177.918,7.258,148.757
C08775=1157.379,209.357,-62.540,-177.915,7.260,148.756
C08776=1157.374,209.627,-62.567,-177.912,7.263,148.756
C08777=1157.369,209.898,-62.594,-177.909,7.266,148.756
C08778=1157.364,210.168,-62.621,-177.906,7.269,148.756
C08779=1157.360,210.439,-62.648,-177.903,7.271,148.756
C08780=1157.355,210.688,-62.673,-177.900,7.274,148.755
C08781=1157.351,210.937,-62.697,-177.897,7.276,148.755
C08782=1157.346,211.186,-62.722,-177.895,7.278,148.755
C08783=1157.341,211.434,-62.747,-177.892,7.281,148.755
C08784=1157.337,211.683,-62.772,-177.889,7.283,148.755
C08785=1157.332,211.932,-62.796,-177.886,7.286,148.754
C08786=1157.328,212.181,-62.821,-177.884,7.288,148.754
C08787=1157.323,212.429,-62.846,-177.881,7.290,148.754
C08788=1157.318,212.678,-62.871,-177.879,7.292,148.754
C08789=1157.314,212.927,-62.895,-177.876,7.295,148.754
C08790=1157.310,213.175,-62.921,-177.873,7.298,148.753
C08791=1157.305,213.424,-62.946,-177.870,7.300,148.753
C08792=1157.301,213.673,-62.970,-177.867,7.303,148.753
C08793=1157.296,213.921,-62.995,-177.865,7.305,148.753
C08794=1157.291,214.170,-63.020,-177.862,7.307,148.752
C08795=1157.287,214.419,-63.046,-177.859,7.309,148.752
C08796=1157.283,214.667,-63.070,-177.857,7.312,148.752
C08797=1157.278,214.917,-63.095,-177.853,7.315,148.752
C08798=1157.273,215.165,-63.120,-177.851,7.317,148.752
C08799=1157.269,215.414,-63.145,-177.848,7.320,148.751
C08800=1157.265,215.662,-63.170,-177.846,7.322,148.751
C08801=1157.260,215.912,-63.195,-177.843,7.325,148.751
C08802=1157.255,216.160,-63.221,-177.840,7.327,148.751
C08803=1157.251,216.409,-63.246,-177.837,7.329,148.751
C08804=1157.247,216.657,-63.270,-177.834,7.332,148.750
C08805=1157.242,216.906,-63.295,-177.832,7.334,148.750
C08806=1157.237,217.154,-63.321,-177.829,7.337,148.750
C08807=1157.233,217.404,-63.346,-177.826,7.340,148.750
C08808=1157.228,217.652,-63.371,-177.824,7.342,148.750
C08809=1157.225,217.900,-63.396,-177.821,7.344,148.750
C08810=1157.219,218.149,-63.421,-177.818,7.346,148.749
C08811=1157.215,218.398,-63.447,-177.816,7.349,148.749
C08812=1157.210,218.647,-63.471,-177.812,7.352,148.749
C08813=1157.206,218.895,-63.497,-177.810,7.354,148.749
C08814=1157.202,219.144,-63.523,-177.807,7.357,148.749
C08815=1157.196,219.393,-63.548,-177.805,7.359,148.748
C08816=1157.193,219.641,-63.573,-177.802,7.362,148.748
C08817=1157.188,219.890,-63.598,-177.799,7.364,148.748
C08818=1157.184,220.139,-63.623,-177.796,7.366,148.748
C08819=1157.179,220.387,-63.649,-177.794,7.369,148.748
C08820=1157.175,220.636,-63.674,-177.790,7.372,148.748
C08821=1157.170,220.885,-63.700,-177.788,7.374,148.747
C08822=1157.165,221.133,-63.725,-177.785,7.377,148.747
C08823=1157.161,221.382,-63.751,-177.782,7.379,148.747
C08824=1157.157,221.631,-63.776,-177.780,7.382,148.747
C08825=1157.152,221.879,-63.802,-177.777,7.384,148.747
C08826=1157.147,222.129,-63.827,-177.774,7.386,148.746
C08827=1157.143,222.377,-63.852,-177.772,7.389,148.746
C08828=1157.138,222.626,-63.878,-177.768,7.392,148.746
C08829=1157.134,222.874,-63.904,-177.766,7.394,148.746
C08830=1157.129,223.122,-63.929,-177.763,7.397,148.746
C08831=1157.125,223.371,-63.955,-177.760,7.399,148.746
C08832=1157.121,223.620,-63.980,-177.758,7.402,148.745
C08833=1157.116,223.869,-64.005,-177.755,7.405,148.745
C08834=1157.112,224.118,-64.031,-177.752,7.407,148.745
C08835=1157.107,224.366,-64.057,-177.750,7.409,148.745
C08836=1157.102,224.614,-64.082,-177.747,7.412,148.745
C08837=1157.098,224.863,-64.108,-177.744,7.415,148.745
C08838=1157.094,225.112,-64.134,-177.742,7.417,148.744
C08839=1157.089,225.360,-64.159,-177.739,7.420,148.744
C08840=1157.085,225.609,-64.185,-177.736,7.422,148.744
C08841=1157.081,225.858,-64.210,-177.733,7.424,148.744
C08842=1157.077,226.107,-64.236,-177.731,7.427,148.744
C08843=1157.071,226.355,-64.262,-177.727,7.430,148.744
C08844=1157.067,226.604,-64.288,-177.725,7.432,148.743
C08845=1157.063,226.853,-64.314,-177.722,7.435,148.743
C08846=1157.058,227.101,-64.339,-177.719,7.438,148.743
C08847=1157.053,227.350,-64.365,-177.717,7.440,148.743
C08848=1157.049,227.598,-64.391,-177.714,7.443,148.743
C08849=1157.045,227.847,-64.416,-177.711,7.446,148.743
C08850=1157.039,228.096,-64.442,-177.709,7.447,148.742
C08851=1157.036,228.344,-64.469,-177.706,7.450,148.742
C08852=1157.031,228.593,-64.494,-177.703,7.453,148.742
C08853=1157.027,228.841,-64.520,-177.700,7.456,148.742
C08854=1157.023,229.090,-64.546,-177.698,7.458,148.742
C08855=1157.017,229.339,-64.572,-177.695,7.461,148.742
C08856=1157.013,229.587,-64.598,-177.692,7.464,148.742
C08857=1157.009,229.836,-64.624,-177.689,7.466,148.741
C08858=1157.005,230.084,-64.650,-177.687,7.469,148.741
C08859=1156.999,230.333,-64.676,-177.684,7.472,148.741
C08860=1156.995,230.582,-64.702,-177.681,7.474,148.741
C08861=1156.991,230.830,-64.727,-177.678,7.476,148.741
C08862=1156.987,231.079,-64.754,-177.676,7.479,148.741
C08863=1156.982,231.328,-64.780,-177.673,7.482,148.741
C08864=1156.978,231.576,-64.806,-177.670,7.484,148.740
C08865=1156.973,231.824,-64.832,-177.667,7.487,148.740
C08866=1156.968,232.073,-64.858,-177.665,7.490,148.740
C08867=1156.964,232.322,-64.884,-177.662,7.493,148.740
C08868=1156.960,232.570,-64.911,-177.659,7.494,148.740
C08869=1156.955,232.819,-64.937,-177.656,7.497,148.740
C08870=1156.951,233.068,-64.963,-177.654,7.500,148.740
C08871=1156.947,233.316,-64.989,-177.651,7.502,148.739
C08872=1156.942,233.565,-65.015,-177.648,7.505,148.739
C08873=1156.937,233.813,-65.041,-177.645,7.508,148.739
C08874=1156.933,234.062,-65.067,-177.643,7.511,148.739
C08875=1156.928,234.311,-65.094,-177.640,7.513,148.739
C08876=1156.924,234.559,-65.120,-177.637,7.516,148.739
C08877=1156.920,234.808,-65.147,-177.634,7.519,148.738
C08878=1156.916,235.056,-65.173,-177.632,7.522,148.738
C08879=1156.911,235.305,-65.199,-177.629,7.524,148.738
C08880=1156.906,235.577,-65.228,-177.626,7.526,148.738
C08881=1156.902,235.848,-65.256,-177.623,7.530,148.738
C08882=1156.896,236.120,-65.286,-177.620,7.533,148.738
C08883=1156.892,236.392,-65.314,-177.617,7.536,148.738
C08884=1156.887,236.640,-65.341,-177.615,7.538,148.737
C08885=1156.883,236.889,-65.367,-177.612,7.541,148.737
C08886=1156.878,237.138,-65.393,-177.609,7.544,148.737
C08887=1156.874,237.386,-65.420,-177.606,7.546,148.737
C08888=1156.869,237.635,-65.446,-177.603,7.549,148.737
C08889=1156.865,237.883,-65.473,-177.601,7.551,148.737
C08890=1156.861,238.132,-65.500,-177.598,7.554,148.737
C08891=1156.857,238.381,-65.526,-177.595,7.557,148.737
C08892=1156.851,238.628,-65.552,-177.592,7.560,148.736
C08893=1156.847,238.877,-65.579,-177.590,7.562,148.736
C08894=1156.842,239.126,-65.605,-177.587,7.565,148.736
C08895=1156.838,239.374,-65.632,-177.584,7.568,148.736
C08896=1156.834,239.622,-65.659,-177.582,7.571,148.736
C08897=1156.829,239.871,-65.685,-177.579,7.573,148.736
C08898=1156.825,240.120,-65.711,-177.576,7.575,148.736
C08899=1156.820,240.368,-65.738,-177.573,7.578,148.736
C08900=1156.816,240.617,-65.765,-177.571,7.581,148.736
C08901=1156.812,240.866,-65.792,-177.568,7.584,148.735
C08902=1156.807,241.115,-65.819,-177.566,7.586,148.735
C08903=1156.803,241.363,-65.845,-177.563,7.589,148.735
C08904=1156.799,241.611,-65.872,-177.560,7.592,148.735
C08905=1156.794,241.860,-65.899,-177.557,7.595,148.735
C08906=1156.790,242.109,-65.925,-177.554,7.598,148.735
C08907=1156.785,242.357,-65.952,-177.552,7.600,148.735
C08908=1156.781,242.606,-65.979,-177.549,7.603,148.735
C08909=1156.777,242.854,-66.006,-177.546,7.606,148.735
C08910=1156.772,243.102,-66.033,-177.543,7.608,148.734
C08911=1156.767,243.351,-66.060,-177.540,7.611,148.734
C08912=1156.763,243.599,-66.086,-177.538,7.613,148.734
C08913=1156.759,243.847,-66.113,-177.535,7.616,148.734
C08914=1156.754,244.097,-66.140,-177.533,7.619,148.734
C08915=1156.749,244.345,-66.167,-177.530,7.622,148.734
C08916=1156.746,244.594,-66.193,-177.527,7.625,148.734
C08917=1156.741,244.842,-66.221,-177.524,7.627,148.734
C08918=1156.736,245.091,-66.248,-177.522,7.630,148.733
C08919=1156.732,245.339,-66.275,-177.519,7.633,148.733
C08920=1156.728,245.588,-66.301,-177.516,7.636,148.733
C08921=1156.723,245.836,-66.328,-177.513,7.639,148.733
C08922=1156.719,246.085,-66.355,-177.511,7.641,148.733
C08923=1156.714,246.332,-66.383,-177.508,7.644,148.733
C08924=1156.711,246.581,-66.410,-177.505,7.647,148.733
C08925=1156.706,246.830,-66.437,-177.503,7.650,148.733
C08926=1156.702,247.078,-66.464,-177.499,7.652,148.733
C08927=1156.697,247.327,-66.491,-177.497,7.655,148.733
C08928=1156.692,247.575,-66.518,-177.495,7.657,148.732
C08929=1156.688,247.824,-66.545,-177.492,7.660,148.732
C08930=1156.684,248.073,-66.573,-177.489,7.663,148.732
C08931=1156.680,248.321,-66.599,-177.486,7.666,148.732
C08932=1156.675,248.569,-66.627,-177.483,7.669,148.732
C08933=1156.671,248.818,-66.654,-177.481,7.672,148.732
C08934=1156.666,249.066,-66.681,-177.478,7.674,148.732
C08935=1156.662,249.315,-66.708,-177.476,7.677,148.732
C08936=1156.657,249.564,-66.735,-177.472,7.680,148.732
C08937=1156.653,249.812,-66.763,-177.470,7.683,148.732
C08938=1156.648,250.060,-66.790,-177.467,7.685,148.732
C08939=1156.644,250.309,-66.817,-177.464,7.688,148.731
C08940=1156.640,250.557,-66.846,-177.461,7.691,148.731
C08941=1156.635,250.806,-66.873,-177.459,7.693,148.731
C08942=1156.631,251.054,-66.899,-177.456,7.696,148.731
C08943=1156.627,251.302,-66.926,-177.454,7.699,148.731
C08944=1156.623,251.551,-66.954,-177.451,7.702,148.731
C08945=1156.618,251.799,-66.981,-177.448,7.705,148.731
C08946=1156.614,252.048,-67.008,-177.445,7.708,148.731
C08947=1156.609,252.296,-67.036,-177.443,7.711,148.731
C08948=1156.605,252.545,-67.064,-177.440,7.713,148.731
C08949=1156.601,252.793,-67.091,-177.438,7.716,148.731
C08950=1156.596,253.041,-67.118,-177.435,7.719,148.731
C08951=1156.592,253.291,-67.146,-177.432,7.722,148.731
C08952=1156.587,253.539,-67.174,-177.429,7.725,148.731
C08953=1156.582,253.787,-67.201,-177.426,7.728,148.730
C08954=1156.578,254.035,-67.229,-177.424,7.731,148.730
C08955=1156.574,254.284,-67.256,-177.421,7.733,148.730
C08956=1156.570,254.532,-67.284,-177.418,7.736,148.730
C08957=1156.565,254.781,-67.311,-177.416,7.739,148.730
C08958=1156.561,255.029,-67.339,-177.413,7.742,148.730
C08959=1156.557,255.278,-67.367,-177.410,7.744,148.730
C08960=1156.552,255.526,-67.394,-177.407,7.747,148.730
C08961=1156.548,255.775,-67.422,-177.404,7.750,148.730
C08962=1156.544,256.023,-67.449,-177.402,7.753,148.730
C08963=1156.539,256.271,-67.478,-177.399,7.756,148.730
C08964=1156.535,256.520,-67.505,-177.397,7.758,148.729
C08965=1156.530,256.768,-67.533,-177.394,7.761,148.729
C08966=1156.526,257.017,-67.560,-177.391,7.764,148.729
C08967=1156.522,257.265,-67.588,-177.388,7.767,148.729
C08968=1156.518,257.513,-67.616,-177.386,7.770,148.729
C08969=1156.513,257.762,-67.644,-177.383,7.773,148.729
C08970=1156.508,258.010,-67.672,-177.380,7.776,148.729
C08971=1156.504,258.258,-67.700,-177.377,7.779,148.729
C08972=1156.500,258.507,-67.727,-177.375,7.782,148.729
C08973=1156.495,258.756,-67.755,-177.372,7.785,148.729
C08974=1156.491,259.004,-67.784,-177.370,7.787,148.729
C08975=1156.487,259.252,-67.811,-177.367,7.790,148.729
C08976=1156.482,259.501,-67.838,-177.364,7.793,148.729
C08977=1156.478,259.749,-67.867,-177.362,7.796,148.729
C08978=1156.473,259.997,-67.895,-177.359,7.799,148.729
C08979=1156.470,260.246,-67.923,-177.356,7.802,148.729
C08980=1156.465,260.494,-67.951,-177.353,7.805,148.729
C08981=1156.460,260.743,-67.979,-177.351,7.808,148.729
C08982=1156.456,260.991,-68.007,-177.348,7.811,148.729
C08983=1156.452,261.240,-68.035,-177.345,7.814,148.728
C08984=1156.448,261.513,-68.065,-177.342,7.817,148.728
C08985=1156.442,261.786,-68.096,-177.340,7.820,148.728
C08986=1156.437,262.059,-68.128,-177.336,7.823,148.728
C08987=1156.433,262.332,-68.158,-177.333,7.826,148.728
C08988=1156.429,262.581,-68.187,-177.331,7.829,148.728
C08989=1156.424,262.829,-68.215,-177.328,7.832,148.728
C08990=1156.420,263.078,-68.242,-177.325,7.835,148.728
C08991=1156.415,263.326,-68.271,-177.322,7.838,148.728
C08992=1156.411,263.575,-68.299,-177.320,7.841,148.728
C08993=1156.407,263.823,-68.327,-177.317,7.843,148.728
C08994=1156.402,264.072,-68.355,-177.315,7.846,148.728
C08995=1156.398,264.319,-68.383,-177.312,7.849,148.728
C08996=1156.393,264.568,-68.412,-177.309,7.852,148.728
C08997=1156.389,264.817,-68.440,-177.306,7.855,148.728
C08998=1156.385,265.064,-68.469,-177.304,7.858,148.728
C08999=1156.381,265.313,-68.497,-177.301,7.861,148.728
C09000=1156.376,265.561,-68.526,-177.298,7.864,148.728
C09001=1156.372,265.810,-68.554,-177.296,7.867,148.728
C09002=1156.368,266.058,-68.582,-177.293,7.870,148.728
C09003=1156.363,266.307,-68.610,-177.290,7.873,148.728
C09004=1156.359,266.554,-68.638,-177.287,7.876,148.728
C09005=1156.354,266.803,-68.667,-177.285,7.879,148.727
C09006=1156.350,267.052,-68.696,-177.282,7.882,148.727
C09007=1156.346,267.299,-68.724,-177.279,7.885,148.727
C09008=1156.341,267.548,-68.753,-177.277,7.888,148.728
C09009=1156.337,267.796,-68.781,-177.274,7.891,148.727
C09010=1156.333,268.045,-68.809,-177.271,7.894,148.727
C09011=1156.329,268.294,-68.837,-177.268,7.897,148.727
C09012=1156.324,268.541,-68.867,-177.266,7.900,148.727
C09013=1156.320,268.790,-68.895,-177.263,7.903,148.727
C09014=1156.315,269.038,-68.923,-177.261,7.905,148.727
C09015=1156.311,269.286,-68.953,-177.258,7.908,148.727
C09016=1156.307,269.535,-68.981,-177.256,7.911,148.727
C09017=1156.302,269.783,-69.009,-177.253,7.914,148.727
C09018=1156.298,270.032,-69.037,-177.250,7.917,148.727
C09019=1156.294,270.280,-69.067,-177.247,7.920,148.727
C09020=1156.289,270.528,-69.095,-177.245,7.923,148.727
C09021=1156.286,270.776,-69.124,-177.242,7.926,148.727
C09022=1156.281,271.025,-69.153,-177.240,7.929,148.727
C09023=1156.276,271.273,-69.181,-177.237,7.932,148.727
C09024=1156.273,271.521,-69.210,-177.234,7.935,148.727
C09025=1156.268,271.770,-69.239,-177.231,7.938,148.727
C09026=1156.263,272.018,-69.268,-177.228,7.941,148.727
C09027=1156.260,272.266,-69.296,-177.226,7.944,148.727
C09028=1156.255,272.515,-69.325,-177.223,7.947,148.727
C09029=1156.250,272.763,-69.354,-177.221,7.950,148.727
C09030=1156.246,273.011,-69.382,-177.218,7.953,148.727
C09031=1156.242,273.259,-69.411,-177.215,7.956,148.727
C09032=1156.238,273.508,-69.440,-177.212,7.959,148.727
C09033=1156.233,273.756,-69.469,-177.210,7.962,148.727
C09034=1156.229,274.004,-69.498,-177.207,7.965,148.727
C09035=1156.225,274.253,-69.527,-177.204,7.968,148.727
C09036=1156.220,274.500,-69.556,-177.202,7.971,148.727
C09037=1156.216,274.749,-69.584,-177.199,7.974,148.727
C09038=1156.212,274.997,-69.614,-177.197,7.977,148.727
C09039=1156.208,275.246,-69.642,-177.194,7.980,148.727
C09040=1156.204,275.494,-69.672,-177.191,7.983,148.727
C09041=1156.199,275.742,-69.701,-177.188,7.986,148.727
C09042=1156.195,275.991,-69.729,-177.186,7.989,148.727
C09043=1156.190,276.239,-69.759,-177.183,7.992,148.727
C09044=1156.186,276.487,-69.788,-177.180,7.995,148.727
C09045=1156.182,276.735,-69.816,-177.178,7.998,148.727
C09046=1156.178,276.983,-69.845,-177.175,8.001,148.727
C09047=1156.174,277.232,-69.875,-177.173,8.005,148.727
C09048=1156.169,277.480,-69.904,-177.170,8.008,148.727
C09049=1156.165,277.729,-69.933,-177.167,8.010,148.727
C09050=1156.161,277.977,-69.963,-177.164,8.013,148.727
C09051=1156.156,278.225,-69.992,-177.162,8.016,148.727
C09052=1156.152,278.473,-70.021,-177.159,8.020,148.727
C09053=1156.147,278.722,-70.050,-177.157,8.023,148.727
C09054=1156.144,278.970,-70.079,-177.154,8.026,148.727
C09055=1156.140,279.218,-70.108,-177.151,8.028,148.727
C09056=1156.135,279.466,-70.138,-177.149,8.032,148.727
C09057=1156.131,279.714,-70.167,-177.145,8.036,148.727
C09058=1156.126,279.962,-70.196,-177.143,8.038,148.727
C09059=1156.122,280.211,-70.225,-177.140,8.042,148.727
C09060=1156.118,280.459,-70.254,-177.137,8.045,148.727
C09061=1156.114,280.708,-70.284,-177.135,8.048,148.727
C09062=1156.109,280.956,-70.313,-177.132,8.051,148.727
C09063=1156.105,281.204,-70.343,-177.130,8.054,148.727
C09064=1156.101,281.452,-70.372,-177.127,8.057,148.727
C09065=1156.096,281.700,-70.401,-177.124,8.060,148.727
C09066=1156.092,281.948,-70.431,-177.122,8.063,148.727
C09067=1156.088,282.196,-70.460,-177.119,8.066,148.727
C09068=1156.083,282.445,-70.490,-177.116,8.069,148.727
C09069=1156.079,282.693,-70.520,-177.114,8.072,148.727
C09070=1156.075,282.942,-70.549,-177.111,8.075,148.727
C09071=1156.070,283.190,-70.579,-177.108,8.078,148.727
C09072=1156.066,283.438,-70.608,-177.106,8.081,148.727
C09073=1156.062,283.686,-70.637,-177.103,8.084,148.727
C09074=1156.058,283.935,-70.667,-177.101,8.087,148.727
C09075=1156.054,284.183,-70.696,-177.098,8.090,148.727
C09076=1156.050,284.431,-70.726,-177.096,8.094,148.727
C09077=1156.046,284.679,-70.756,-177.093,8.097,148.727
C09078=1156.041,284.927,-70.786,-177.090,8.099,148.727
C09079=1156.037,285.176,-70.816,-177.087,8.104,148.728
C09080=1156.032,285.423,-70.845,-177.084,8.106,148.727
C09081=1156.028,285.671,-70.874,-177.082,8.109,148.727
C09082=1156.023,285.920,-70.904,-177.079,8.113,148.728
C09083=1156.019,286.168,-70.934,-177.077,8.116,148.728
C09084=1156.015,286.416,-70.964,-177.074,8.119,148.728
C09085=1156.010,286.664,-70.993,-177.071,8.122,148.728
C09086=1156.006,286.913,-71.023,-177.069,8.125,148.728
C09087=1156.002,287.160,-71.053,-177.066,8.128,148.728
C09088=1155.998,287.436,-71.086,-177.063,8.132,148.728
C09089=1155.993,287.711,-71.119,-177.060,8.135,148.728
C09090=1155.988,287.986,-71.152,-177.057,8.139,148.728
C09091=1155.983,288.261,-71.186,-177.055,8.142,148.728
C09092=1155.979,288.510,-71.215,-177.052,8.145,148.728
C09093=1155.975,288.758,-71.245,-177.049,8.148,148.728
C09094=1155.971,289.006,-71.275,-177.047,8.151,148.728
C09095=1155.966,289.254,-71.305,-177.043,8.155,148.728
C09096=1155.962,289.502,-71.335,-177.041,8.158,148.728
C09097=1155.958,289.750,-71.364,-177.038,8.161,148.728
C09098=1155.953,289.999,-71.394,-177.036,8.164,148.728
C09099=1155.950,290.247,-71.425,-177.033,8.167,148.728
C09100=1155.946,290.495,-71.454,-177.031,8.170,148.728
C09101=1155.941,290.743,-71.485,-177.028,8.173,148.728
C09102=1155.937,290.992,-71.515,-177.025,8.177,148.728
C09103=1155.933,291.239,-71.545,-177.023,8.179,148.728
C09104=1155.928,291.488,-71.575,-177.020,8.183,148.729
C09105=1155.924,291.735,-71.605,-177.018,8.186,148.729
C09106=1155.920,291.984,-71.634,-177.014,8.189,148.729
C09107=1155.915,292.232,-71.665,-177.012,8.193,148.729
C09108=1155.912,292.481,-71.695,-177.009,8.196,148.729
C09109=1155.907,292.729,-71.726,-177.007,8.199,148.729
C09110=1155.903,292.976,-71.756,-177.004,8.202,148.729
C09111=1155.898,293.225,-71.786,-177.002,8.205,148.729
C09112=1155.894,293.472,-71.816,-176.999,8.208,148.729
C09113=1155.890,293.721,-71.846,-176.996,8.211,148.729
C09114=1155.886,293.969,-71.876,-176.994,8.214,148.729
C09115=1155.882,294.217,-71.907,-176.991,8.218,148.729
C09116=1155.877,294.466,-71.937,-176.988,8.221,148.729
C09117=1155.874,294.713,-71.967,-176.986,8.224,148.729
C09118=1155.869,294.961,-71.998,-176.983,8.228,148.729
C09119=1155.865,295.209,-72.027,-176.981,8.231,148.729
C09120=1155.861,295.458,-72.058,-176.978,8.234,148.730
C09121=1155.857,295.706,-72.089,-176.975,8.237,148.730
C09122=1155.852,295.954,-72.119,-176.973,8.240,148.729
C09123=1155.848,296.202,-72.149,-176.970,8.244,148.730
C09124=1155.843,296.450,-72.180,-176.967,8.247,148.730
C09125=1155.840,296.698,-72.210,-176.965,8.250,148.730
C09126=1155.836,296.946,-72.241,-176.962,8.253,148.730
C09127=1155.831,297.194,-72.272,-176.960,8.256,148.730
C09128=1155.827,297.443,-72.301,-176.957,8.259,148.730
C09129=1155.823,297.691,-72.332,-176.955,8.263,148.730
C09130=1155.819,297.939,-72.362,-176.951,8.266,148.730
C09131=1155.814,298.187,-72.393,-176.949,8.270,148.730
C09132=1155.810,298.435,-72.424,-176.946,8.273,148.730
C09133=1155.806,298.683,-72.455,-176.944,8.276,148.730
C09134=1155.802,298.931,-72.485,-176.941,8.279,148.730
C09135=1155.797,299.179,-72.516,-176.939,8.282,148.731
C09136=1155.793,299.427,-72.546,-176.936,8.285,148.731
C09137=1155.789,299.675,-72.577,-176.933,8.289,148.731
C09138=1155.784,299.924,-72.607,-176.930,8.292,148.731
C09139=1155.780,300.172,-72.638,-176.928,8.295,148.731
C09140=1155.776,300.420,-72.669,-176.925,8.298,148.731
C09141=1155.772,300.668,-72.699,-176.923,8.302,148.731
C09142=1155.768,300.916,-72.730,-176.920,8.305,148.731
C09143=1155.764,301.164,-72.761,-176.918,8.308,148.731
C09144=1155.760,301.412,-72.792,-176.915,8.312,148.731
C09145=1155.755,301.660,-72.823,-176.912,8.315,148.731
C09146=1155.752,301.908,-72.854,-176.910,8.318,148.732
C09147=1155.747,302.156,-72.884,-176.907,8.321,148.732
C09148=1155.743,302.404,-72.915,-176.905,8.324,148.732
C09149=1155.739,302.653,-72.946,-176.902,8.327,148.732
